# B&R Automation Studio project NAINV104C00R8L515F00 (part 16)

#### Visu_Page.typ - Change By Project
```iecst
(*2020-10-08*)
(**)
(*Page*)

TYPE
	tyUIP0000SSaver : 	STRUCT
		tySSaver : tyLyrP0000SSaver := (tyTxtMcStat:=(usiValueIdx:=3));
		tyMsgBoxHide : tyLyrC0008MsgBox := (tyBitmapIcon:=(uiRtStat:=1),tyBtnNo:=(uiRtStat:=1),tyBtnYes:=(uiRtStat:=1),tyLyr:=(uiRtStat:=1),tyTxtMsg:=(uiRtStat:=1),tyTxtTitle:=(uiRtStat:=1));
		tyMsgBoxLoginAsk : tyLyrC0008MsgBox := (tyBitmapIcon:=(usiValueIdx:=1),tyTxtTitle:=(usiValueIdx:=1),tyTxtMsg:=(usiValueIdx:=173),tyBtnYes:=(usiBitmapIdx:=1,usiTxtIdx:=3),tyBtnNo:=(usiBitmapIdx:=4,usiTxtIdx:=6),tyLyr:=(uiRtStat:=0));
	END_STRUCT;
END_TYPE

(**)

TYPE
	tyUIP0001Startup : 	STRUCT
		tyStartup : tyLyrP0001Startup;
		tyInitial : tyLyrP0001Initial;
		tyMsgBoxHide : tyLyrC0008MsgBox := (tyBitmapIcon:=(uiRtStat:=1),tyBtnNo:=(uiRtStat:=1),tyBtnYes:=(uiRtStat:=1),tyLyr:=(uiRtStat:=1),tyTxtMsg:=(uiRtStat:=1),tyTxtTitle:=(uiRtStat:=1));
		tyMsgBoxIPConfig : tyLyrC0008MsgBox := (tyBitmapIcon:=(usiValueIdx:=1),tyBtnNo:=(usiBitmapIdx:=3,usiTxtIdx:=2),tyBtnYes:=(usiBitmapIdx:=1,usiTxtIdx:=1),tyTxtTitle:=(usiValueIdx:=25));
	END_STRUCT;
END_TYPE

(**)

TYPE
	tyUIP0002Menu : 	STRUCT
		tyMenu : tyLyrP0002Menu := (tyBtnAlm:=(uiMaskRtStat:=0),tyBtnCommCtrl:=(uiMaskRtStat:=0),tyBtnGenInput:=(uiMaskRtStat:=0),tyBtnGenOutput:=(uiMaskRtStat:=0),tyBtnLang:=(uiMaskRtStat:=0),tyBtnLFCtrl:=(uiMaskRtStat:=0),tyBtnLFSet:=(uiMaskRtStat:=0),tyBtnMcInfo:=(uiMaskRtStat:=0),tyBtnMcSet:=(uiMaskRtStat:=0),tyBtnMnlRst:=(uiRtStat:=1),tyBtnMovCtrl:=(uiMaskRtStat:=0),tyBtnOpt:=(uiMaskRtStat:=0),tyBtnProdSel:=(uiMaskRtStat:=0),tyBtnProdSet:=(uiMaskRtStat:=0),tyBtnSimu:=(uiMaskRtStat:=0,uiRtStat:=1),tyBtnUsrMgmt:=(uiMaskRtStat:=0),tyGenMaskLyr:=(uiRtStat:=1),tySetMaskLyr:=(uiRtStat:=1));
		tyMsgBoxHide : tyLyrC0008MsgBox := (tyBitmapIcon:=(uiRtStat:=1),tyBtnNo:=(uiRtStat:=1),tyBtnYes:=(uiRtStat:=1),tyTxtMsg:=(uiRtStat:=1),tyTxtTitle:=(uiRtStat:=1),tyLyr:=(uiRtStat:=1));
		tyMsgBoxSelRcpWaitingBrd : tyLyrC0008MsgBox := (tyBitmapIcon:=(usiValueIdx:=1),tyTxtTitle:=(usiValueIdx:=2),tyTxtMsg:=(usiValueIdx:=100),tyBtnYes:=(uiRtStat:=1,usiBitmapIdx:=1,usiTxtIdx:=1),tyBtnNo:=(usiBitmapIdx:=1,usiTxtIdx:=3),tyLyr:=(uiRtStat:=0));
	END_STRUCT;
END_TYPE

(**)

TYPE
	tyUIP0100Login : 	STRUCT
		tyLogin : tyLyrP0100Login := (tyStringPw:=(sKeypadTitle:='Password'),tyStringUsrNm:=(sKeypadTitle:='User Name'));
		tyLogout : tyLyrP0100Logout := (tyLyr:=(uiRtStat:=1));
		tyMsgBoxHide : tyLyrC0008MsgBox := (tyBitmapIcon:=(uiRtStat:=1),tyBtnNo:=(uiRtStat:=1),tyBtnYes:=(uiRtStat:=1),tyTxtMsg:=(uiRtStat:=1),tyTxtTitle:=(uiRtStat:=1),tyLyr:=(uiRtStat:=1));
		tyMsgBoxNmNotExist : tyLyrC0008MsgBox := (tyBitmapIcon:=(usiValueIdx:=1),tyBtnNo:=(usiBitmapIdx:=1,usiTxtIdx:=3),tyBtnYes:=(uiRtStat:=1),tyLyr:=(uiRtStat:=0),tyTxtMsg:=(usiValueIdx:=23),tyTxtTitle:=(usiValueIdx:=1));
		tyMsgBoxPwMismatch : tyLyrC0008MsgBox := (tyBitmapIcon:=(usiValueIdx:=1),tyBtnNo:=(usiBitmapIdx:=1,usiTxtIdx:=3),tyBtnYes:=(uiRtStat:=1),tyLyr:=(uiRtStat:=0),tyTxtMsg:=(usiValueIdx:=24),tyTxtTitle:=(usiValueIdx:=1));
	END_STRUCT;
END_TYPE

(**)

TYPE
	tyUIP0200OpsGen : 	STRUCT
		tyOps : tyLyrP0200OpsGen := (tyBitmapDSCommIcon:=(uiMaskRtStat:=0),tyBitmapUSCommIcon:=(uiMaskRtStat:=0),tyBitmapRlsNewProd:=(uiRtStat:=1),tyBtnRlsNewProd:=(uiRtStat:=1));
		tyUSVSMEMA : tyLyrP0200OpsUSVSMEMA := (tyBtnUBAStat:=(uiRtStat:=1),tyBtnDual:=(uiRtStat:=1),tyLyr:=(uiRtStat:=1));
		tyDSVSMEMA : tyLyrP0200OpsDSVSMEMA := (tyBtnDSBStat:=(uiRtStat:=1),tyBtnDual:=(uiRtStat:=1),tyLyr:=(uiRtStat:=1));
		tyUSVSMEMA1 : tyLyrP0200OpsUSVSMEMA1 := (tyBtnUBAStat:=(uiRtStat:=1),tyBtnDual:=(uiRtStat:=1),tyLyr:=(uiRtStat:=1));
		tyDSVSMEMA1 : tyLyrP0200OpsDSVSMEMA1 := (tyBtnDSBStat:=(uiRtStat:=1),tyBtnDual:=(uiRtStat:=1),tyLyr:=(uiRtStat:=1));
		tyUSVSMEMA2 : tyLyrP0200OpsUSVSMEMA2 := (tyBtnUBAStat:=(uiRtStat:=1),tyBtnDual:=(uiRtStat:=1),tyLyr:=(uiRtStat:=1));
		tyBypsInitConv : tyLyrP0200OpsBypsInitConv := (tyLyr:=(uiRtStat:=1));
		tyMsgBoxHide : tyLyrC0008MsgBox := (tyBitmapIcon:=(uiRtStat:=1),tyBtnNo:=(uiRtStat:=1),tyBtnYes:=(uiRtStat:=1),tyTxtMsg:=(uiRtStat:=1),tyTxtTitle:=(uiRtStat:=1),tyLyr:=(uiRtStat:=1));
		tyMsgBoxRcpSelMsg : tyLyrC0008MsgBox;
		tyMsgBoxRstWaitingBrdAsk : tyLyrC0008MsgBox := (tyBitmapIcon:=(usiValueIdx:=1),tyTxtTitle:=(usiValueIdx:=23),tyTxtMsg:=(usiValueIdx:=125),tyBtnYes:=(usiBitmapIdx:=1,usiTxtIdx:=1),tyBtnNo:=(usiBitmapIdx:=3,usiTxtIdx:=2),tyLyr:=(uiRtStat:=0));
		tyRcyMsgHide : tyLyrC0010RcyMsg := (tyHotspotClose:=(uiRtStat:=1),tyLyr:=(uiRtStat:=1));
		tyRcyMsg : tyLyrC0010RcyMsg;
	END_STRUCT;
END_TYPE

(**)

TYPE
	tyUIP0201OpsConv : 	STRUCT
		tyOps : tyLyrP0201OpsConv := (tyBitmapRlsNewProd:=(uiRtStat:=1),tyBtnRlsNewProd:=(uiRtStat:=1));
		tyIOMonitor : tyLyrP0201OpsConvIOMonitor := (tyLyr:=(uiRtStat:=1));
		tyIOMonitorXStd : tyLyrP0201OpsConvIOMonitorXStd := (tyLyr:=(uiRtStat:=1));
		tyIOMonitorXStdMachineSafety : tyLyrP0201OpsConvIOMonitorMSafe;
		tyBypsInitConv : tyLyrP0200OpsBypsInitConv := (tyLyr:=(uiRtStat:=1));
		tyChgParam : tyLyrP0201OpsConvChgParam := (tyNumProdWidth:=(sKeypadTitle:='Product Width'),tyLyr:=(uiRtStat:=1));
		tyChgParamBkUp : tyLyrP0201OpsConvChgParam;
		tyNaviHide : tyLyrC0004Navi := (tyBtnLeft:=(uiRtStat:=1),tyBtnRgt:=(uiRtStat:=1),tyBtnBack:=(uiRtStat:=1));
		tyNaviBack : tyLyrC0004Navi := (tyBtnLeft:=(uiRtStat:=1),tyBtnRgt:=(uiRtStat:=1),tyBitmapPageDisp:=(uiRtStat:=1));
		tyMsgBoxHide : tyLyrC0008MsgBox := (tyBitmapIcon:=(uiRtStat:=1),tyBtnNo:=(uiRtStat:=1),tyBtnYes:=(uiRtStat:=1),tyTxtMsg:=(uiRtStat:=1),tyTxtTitle:=(uiRtStat:=1),tyLyr:=(uiRtStat:=1));
		tyMsgBoxSaveErr : tyLyrC0008MsgBox := (tyBitmapIcon:=(usiValueIdx:=1),tyTxtTitle:=(usiValueIdx:=7),tyTxtMsg:=(usiValueIdx:=71),tyBtnYes:=(uiRtStat:=1),tyBtnNo:=(usiBitmapIdx:=1,usiTxtIdx:=3));
		tyRcpPopUp : tyLyrC0012RcpPopUp := (tyLyr:=(uiRtStat:=1));
	END_STRUCT;
END_TYPE

(**)

TYPE
	tyUIP0300McInfo : 	STRUCT
		tyMcInfo : tyLyrP0300McInfo;
		tyMsgBoxHide : tyLyrC0008MsgBox := (tyBitmapIcon:=(uiRtStat:=1),tyTxtTitle:=(uiRtStat:=1),tyTxtMsg:=(uiRtStat:=1),tyBtnYes:=(uiRtStat:=1),tyBtnNo:=(uiRtStat:=1),tyLyr:=(uiRtStat:=1));
	END_STRUCT;
END_TYPE

(**)

TYPE
	tyUIP0400ProdSel : 	STRUCT
		tyProdSel : tyLyrP0400ProdSel := (tyStringSearch:=(sKeypadTitle:='Search Keyword'),tyTableRecipe:=(a_tyHotspot:=[(bRtCompl:=TRUE,bValue:=TRUE),14((0))],a_tyStringDataCol0:=[(sValue:='1'),(sValue:='2'),(sValue:='3'),(sValue:='4'),(sValue:='5'),(sValue:='6'),(sValue:='7'),(sValue:='8'),(sValue:='9'),2((sValue:='10')),4((0))],a_tyStringDataCol1:=[(usiColor:=1),14((0))],a_tyStringDataCol2:=[(usiColor:=1),14((0))],tyUISlider:=(iMaxValue:=1991,iMinValue:=1,iValue:=1),tyStringTitle0Col0Row0:=(sValue:='No'),tyStringTitle1Col1Row0:=(sValue:='Program Name'),tyStringTitle2Col2Row0:=(sValue:='Width')));
		tyRcpDet : tyLyrP0400RcpDet := (tyLyr:=(uiRtStat:=1));
		tyMsgBoxHide : tyLyrC0008MsgBox := (tyBitmapIcon:=(uiRtStat:=1),tyBtnNo:=(uiRtStat:=1),tyBtnYes:=(uiRtStat:=1),tyTxtMsg:=(uiRtStat:=1),tyTxtTitle:=(uiRtStat:=1),tyLyr:=(uiRtStat:=1));
		tyMsgBoxListErr : tyLyrC0008MsgBox := (tyBitmapIcon:=(usiValueIdx:=1),tyBtnNo:=(usiBitmapIdx:=1,usiTxtIdx:=3),tyBtnYes:=(uiRtStat:=1),tyLyr:=(uiRtStat:=0),tyTxtMsg:=(usiValueIdx:=42),tyTxtTitle:=(usiValueIdx:=2));
		tyMsgBoxRcpParamErr : tyLyrC0008MsgBox;
		tyMsgBoxLoadErr : tyLyrC0008MsgBox := (tyBitmapIcon:=(usiValueIdx:=1),tyBtnNo:=(usiBitmapIdx:=1,usiTxtIdx:=3),tyBtnYes:=(uiRtStat:=1),tyLyr:=(uiRtStat:=0),tyTxtMsg:=(usiValueIdx:=41),tyTxtTitle:=(usiValueIdx:=2));
		tyMsgBoxSelRcpAsk : tyLyrC0008MsgBox := (tyBitmapIcon:=(usiValueIdx:=1),tyBtnNo:=(usiBitmapIdx:=3,usiTxtIdx:=2),tyBtnYes:=(usiBitmapIdx:=1,usiTxtIdx:=1),tyLyr:=(uiRtStat:=0),tyTxtMsg:=(usiValueIdx:=43),tyTxtTitle:=(usiValueIdx:=2));
		tyMsgBoxSelRcpNoNm : tyLyrC0008MsgBox := (tyBitmapIcon:=(usiValueIdx:=1),tyBtnNo:=(usiBitmapIdx:=1,usiTxtIdx:=3),tyBtnYes:=(uiRtStat:=1),tyLyr:=(uiRtStat:=0),tyTxtMsg:=(usiValueIdx:=44),tyTxtTitle:=(usiValueIdx:=2));
		tyMsgBoxSaveErr : tyLyrC0008MsgBox := (tyBitmapIcon:=(usiValueIdx:=1),tyBtnNo:=(usiBitmapIdx:=1,usiTxtIdx:=3),tyBtnYes:=(uiRtStat:=1),tyLyr:=(uiRtStat:=0),tyTxtMsg:=(usiValueIdx:=71),tyTxtTitle:=(usiValueIdx:=2));
		tyMsgBoxGoToLFCtrlAsk : tyLyrC0008MsgBox := (tyBitmapIcon:=(usiValueIdx:=1),tyTxtTitle:=(usiValueIdx:=2),tyTxtMsg:=(usiValueIdx:=163),tyBtnYes:=(usiBitmapIdx:=1,usiTxtIdx:=1),tyBtnNo:=(usiBitmapIdx:=3,usiTxtIdx:=2),tyLyr:=(uiRtStat:=0));
		tyRcpPopUp : tyLyrC0012RcpPopUp := (tyLyr:=(uiRtStat:=1));
	END_STRUCT;
END_TYPE

(**)

TYPE
	tyUIP0600Alm : 	STRUCT
		tyAlm : tyLyrP0600Alm := (tyBtnCurr:=(bValue:=TRUE));
		tyMsgBoxHide : tyLyrC0008MsgBox := (tyBitmapIcon:=(uiRtStat:=1),tyBtnNo:=(uiRtStat:=1),tyBtnYes:=(uiRtStat:=1),tyTxtMsg:=(uiRtStat:=1),tyTxtTitle:=(uiRtStat:=1),tyLyr:=(uiRtStat:=1));
		tyRcyMsg : tyLyrC0010RcyMsg;
		tyRcyMsgHide : tyLyrC0010RcyMsg := (tyLyr:=(uiRtStat:=1));
		tyBtnCurr : tyUIBtn;
		tyBtnHistory : tyUIBtn;
		tyAlarm : tyUIAlarm;
	END_STRUCT;
END_TYPE

(**)

TYPE
	tyUIP0700LFCtrl : 	STRUCT
		tyLdr : tyLyrP0700LFCtrl := (tyBtnChgSeqAuto:=(uiMaskRtStat:=1),tyBtnChgSeqMnl:=(uiMaskRtStat:=1),tyTable1List:=(a_tyHotspot:=[(bRtCompl:=TRUE,bValue:=TRUE),14(0)],a_tyStringDataCol0:=[(sValue:='1'),(sValue:='2'),(sValue:='3'),(sValue:='4'),(sValue:='5'),(sValue:='6'),(sValue:='7'),(sValue:='8'),(sValue:='9'),(sValue:='10'),(sValue:='11'),(sValue:='12'),3((0))],a_tyStringDataCol1:=[0,14((0))],a_tyStringDataCol2:=[0,14((0))],a_tyStringDataCol4:=[(usiColor:=0),14((0))],a_tyTxtDataCol3:=[(usiColor:=1),14((0))],tyStringTitle0Col0Row0:=(sValue:='No'),tyStringTitle1Col1Row0:=(sValue:='Machine Name'),tyStringTitle2Col2Row0:=(sValue:='IP Address'),tyStringTitle3Col3Row0:=(sValue:='Status'),tyStringTitle4Col4Row0:=(sValue:='Recipe No'),tyUISlider:=(iMaxValue:=50,iMinValue:=1,iValue:=1,uiRtStat:=0)),tyLyr:=(uiRtStat:=0));
		tyMsgBoxHide : tyLyrC0008MsgBox := (tyBitmapIcon:=(uiRtStat:=1),tyBtnNo:=(uiRtStat:=1),tyBtnYes:=(uiRtStat:=1),tyTxtMsg:=(uiRtStat:=1),tyTxtTitle:=(uiRtStat:=1),tyLyr:=(uiRtStat:=1));
		tyMsgBoxChgAllAsk : tyLyrC0008MsgBox := (tyBitmapIcon:=(usiValueIdx:=1),tyTxtTitle:=(usiValueIdx:=9),tyTxtMsg:=(usiValueIdx:=156),tyBtnYes:=(usiBitmapIdx:=1,usiTxtIdx:=1),tyBtnNo:=(usiBitmapIdx:=3,usiTxtIdx:=2));
		tyMsgBoxChgSeqAutoAsk : tyLyrC0008MsgBox := (tyBitmapIcon:=(usiValueIdx:=1),tyTxtTitle:=(usiValueIdx:=9),tyTxtMsg:=(usiValueIdx:=157),tyBtnYes:=(usiBitmapIdx:=1,usiTxtIdx:=1),tyBtnNo:=(usiBitmapIdx:=3,usiTxtIdx:=2));
		tyMsgBoxChgSeqMnlAsk : tyLyrC0008MsgBox := (tyBitmapIcon:=(usiValueIdx:=1),tyTxtTitle:=(usiValueIdx:=9),tyTxtMsg:=(usiValueIdx:=158),tyBtnYes:=(usiBitmapIdx:=1,usiTxtIdx:=1),tyBtnNo:=(usiBitmapIdx:=3,usiTxtIdx:=2));
		tyMsgBoxSyncPLCTmAsk : tyLyrC0008MsgBox := (tyBitmapIcon:=(usiValueIdx:=1),tyTxtTitle:=(usiValueIdx:=9),tyTxtMsg:=(usiValueIdx:=159),tyBtnYes:=(usiBitmapIdx:=1,usiTxtIdx:=1),tyBtnNo:=(usiBitmapIdx:=3,usiTxtIdx:=2));
		tyMsgBoxTerminateOpsAsk : tyLyrC0008MsgBox := (tyBitmapIcon:=(usiValueIdx:=1),tyTxtTitle:=(usiValueIdx:=9),tyTxtMsg:=(usiValueIdx:=160),tyBtnYes:=(usiBitmapIdx:=1,usiTxtIdx:=1),tyBtnNo:=(usiBitmapIdx:=3,usiTxtIdx:=2));
		tyMsgBoxErrorAsk : tyLyrC0008MsgBox := (tyBitmapIcon:=(usiValueIdx:=1),tyTxtTitle:=(usiValueIdx:=9),tyTxtMsg:=(usiValueIdx:=165),tyBtnYes:=(uiRtStat:=1),tyBtnNo:=(usiBitmapIdx:=1,usiTxtIdx:=3));
	END_STRUCT;
END_TYPE

(**)

TYPE
	tyUIP0900GenIn : 	STRUCT
		tyGenIn : tyLyrP0900GenIn;
		tyMsgBoxHide : tyLyrC0008MsgBox := (tyBitmapIcon:=(uiRtStat:=1),tyBtnNo:=(uiRtStat:=1),tyBtnYes:=(uiRtStat:=1),tyTxtMsg:=(uiRtStat:=1),tyTxtTitle:=(uiRtStat:=1),tyLyr:=(uiRtStat:=1));
	END_STRUCT;
END_TYPE

(**)

TYPE
	tyUIP0910GenOut : 	STRUCT
		tyGenOut : tyLyrP0910GenOut;
		tyMsgBoxHide : tyLyrC0008MsgBox := (tyBitmapIcon:=(uiRtStat:=1),tyBtnNo:=(uiRtStat:=1),tyBtnYes:=(uiRtStat:=1),tyTxtMsg:=(uiRtStat:=1),tyTxtTitle:=(uiRtStat:=1),tyLyr:=(uiRtStat:=1));
	END_STRUCT;
END_TYPE

(**)

TYPE
	tyUIP0920MtrNPneuCtrl : 	STRUCT
		tyMtrNPneuCtrl : tyLyrP0920MtrNPneuCtrl;
		tyFullMaskHide : tyLyrC0002FullMask := (tyLyr:=(uiRtStat:=1));
		tyFullMaskEStop : tyLyrC0002FullMask := (tyBtnMask:=(usiTxtIdx:=20),tyLyr:=(uiRtStat:=0));
		tyFullMaskCWSig : tyLyrC0002FullMask := (tyBtnMask:=(usiTxtIdx:=21),tyLyr:=(uiRtStat:=0));
		tyFullMaskSafetyRly : tyLyrC0002FullMask := (tyBtnMask:=(usiTxtIdx:=12),tyLyr:=(uiRtStat:=0));
		tyMsgBoxHide : tyLyrC0008MsgBox := (tyBitmapIcon:=(uiRtStat:=1),tyBtnNo:=(uiRtStat:=1),tyBtnYes:=(uiRtStat:=1),tyTxtMsg:=(uiRtStat:=1),tyTxtTitle:=(uiRtStat:=1),tyLyr:=(uiRtStat:=1));
	END_STRUCT;
END_TYPE

(**)

TYPE
	tyUIP0921ClampNoRS : 	STRUCT
		tyCom : tyLyrP0921ClampNoRSCom;
		tyDC : tyLyrP0921ClampNoRSDC := (tyLyr:=(uiRtStat:=1));
		tyFB : tyLyrP0921ClampNoRSFB;
		tyFullMaskHide : tyLyrC0002FullMask := (tyLyr:=(uiRtStat:=1));
		tyFullMaskEStop : tyLyrC0002FullMask := (tyBtnMask:=(usiTxtIdx:=20),tyLyr:=(uiRtStat:=0));
		tyFullMaskCWSig : tyLyrC0002FullMask := (tyBtnMask:=(usiTxtIdx:=21),tyLyr:=(uiRtStat:=0));
		tyFullMaskSafetyRly : tyLyrC0002FullMask := (tyBtnMask:=(usiTxtIdx:=12),tyLyr:=(uiRtStat:=0));
		tyNaviBack : tyLyrC0004Navi := (tyBtnLeft:=(uiRtStat:=1),tyBtnRgt:=(uiRtStat:=1),tyBtnBack:=(uiRtStat:=0));
		tyMsgBoxHide : tyLyrC0008MsgBox := (tyBitmapIcon:=(uiRtStat:=1),tyBtnNo:=(uiRtStat:=1),tyBtnYes:=(uiRtStat:=1),tyTxtMsg:=(uiRtStat:=1),tyTxtTitle:=(uiRtStat:=1),tyLyr:=(uiRtStat:=1));
	END_STRUCT;
END_TYPE

(**)

TYPE
	tyUIP0922InletNOutletShutter : 	STRUCT
		tyInletShutterCom : tyLyrP0922InletShutterCom;
		tyInletShutterDC : tyLyrP0922InletShutterDC := (tyLyr:=(uiRtStat:=1));
		tyInletShutterFB : tyLyrP0922InletShutterFB;
		tyInletShutterDis : tyLyrP0922InletShutterDis := (tyLyr:=(uiRtStat:=1));
		tyOutletShutterCom : tyLyrP0922OutletShutterCom;
		tyOutletShutterDC : tyLyrP0922OutletShutterDC := (tyLyr:=(uiRtStat:=1));
		tyOutletShutterFB : tyLyrP0922OutletShutterFB;
		tyOutletShutterDis : tyLyrP0922OutletShutterDis := (tyLyr:=(uiRtStat:=1));
		tyDualMaskHide : tyLyrC0003DualMask := (tyLyr:=(uiRtStat:=1));
		tyDualMaskEStop : tyLyrC0003DualMask := (tyBtnLeftMask:=(uiMaskRtStat:=0,usiTxtIdx:=20),tyBtnRgtMask:=(uiMaskRtStat:=0,usiTxtIdx:=20));
		tyDualMaskCWSig : tyLyrC0003DualMask := (tyBtnLeftMask:=(uiMaskRtStat:=0,usiTxtIdx:=21),tyBtnRgtMask:=(uiMaskRtStat:=0,usiTxtIdx:=21));
		tyDualMaskSafetyRly : tyLyrC0003DualMask := (tyBtnLeftMask:=(uiMaskRtStat:=0,usiTxtIdx:=12),tyBtnRgtMask:=(uiMaskRtStat:=0,usiTxtIdx:=12));
		tyDualMaskAWMovInterrupt : tyLyrC0003DualMask := (tyBtnLeftMask:=(uiMaskRtStat:=0,usiTxtIdx:=17),tyBtnRgtMask:=(uiMaskRtStat:=0,usiTxtIdx:=17));
		tyNaviBack : tyLyrC0004Navi := (tyBtnLeft:=(uiRtStat:=1),tyBtnRgt:=(uiRtStat:=1),tyBtnBack:=(uiRtStat:=0));
		tyMsgBoxHide : tyLyrC0008MsgBox := (tyBitmapIcon:=(uiRtStat:=1),tyBtnNo:=(uiRtStat:=1),tyBtnYes:=(uiRtStat:=1),tyLyr:=(uiRtStat:=1),tyTxtMsg:=(uiRtStat:=1),tyTxtTitle:=(uiRtStat:=1));
	END_STRUCT;
END_TYPE

(**)

TYPE
	tyUIP0923Stopper : 	STRUCT
		tyCom : tyLyrP0923StopperCom;
		tyDC : tyLyrP0923StopperDC := (tyLyr:=(uiRtStat:=1));
		tyFB : tyLyrP0923StopperFB;
		tyFullMaskHide : tyLyrC0002FullMask := (tyLyr:=(uiRtStat:=1));
		tyFullMaskEStop : tyLyrC0002FullMask := (tyBtnMask:=(usiTxtIdx:=20),tyLyr:=(uiRtStat:=0));
		tyFullMaskCWSig : tyLyrC0002FullMask := (tyBtnMask:=(usiTxtIdx:=21),tyLyr:=(uiRtStat:=0));
		tyFullMaskSafetyRly : tyLyrC0002FullMask := (tyBtnMask:=(usiTxtIdx:=12),tyLyr:=(uiRtStat:=0));
		tyNaviBack : tyLyrC0004Navi := (tyBtnLeft:=(uiRtStat:=1),tyBtnRgt:=(uiRtStat:=1),tyBtnBack:=(uiRtStat:=0));
		tyMsgBoxHide : tyLyrC0008MsgBox := (tyBitmapIcon:=(uiRtStat:=1),tyBtnNo:=(uiRtStat:=1),tyBtnYes:=(uiRtStat:=1),tyTxtMsg:=(uiRtStat:=1),tyTxtTitle:=(uiRtStat:=1),tyLyr:=(uiRtStat:=1));
	END_STRUCT;
END_TYPE

(**)

TYPE
	tyUIP0924ClampWithRS : 	STRUCT
		tyClamp1WithRSCom : tyLyrP0924Clamp1WithRSCom;
		tyClamp1WithRSDC : tyLyrP0924Clamp1WithRSDC := (tyLyr:=(uiRtStat:=1));
		tyClamp1WithRSFB : tyLyrP0924Clamp1WithRSFB;
		tyClamp1WithRSDis : tyLyrP0924Clamp1WithRSDis := (tyLyr:=(uiRtStat:=1));
		tyClamp2WithRSCom : tyLyrP0924Clamp2WithRSCom;
		tyClamp2WithRSDC : tyLyrP0924Clamp2WithRSDC := (tyLyr:=(uiRtStat:=1));
		tyClamp2WithRSFB : tyLyrP0924Clamp2WithRSFB;
		tyClamp2WithRSDis : tyLyrP0924Clamp2WithRSDis := (tyLyr:=(uiRtStat:=1));
		tyClamp3WithRSCom : tyLyrP0924Clamp3WithRSCom;
		tyClamp3WithRSDC : tyLyrP0924Clamp3WithRSDC := (tyLyr:=(uiRtStat:=1));
		tyClamp3WithRSFB : tyLyrP0924Clamp3WithRSFB;
		tyClamp3WithRSDis : tyLyrP0924Clamp3WithRSDis := (tyLyr:=(uiRtStat:=1));
		tyDualMaskHide : tyLyrC0003DualMask := (tyLyr:=(uiRtStat:=1));
		tyDualMaskEStop : tyLyrC0003DualMask := (tyBtnLeftMask:=(uiMaskRtStat:=0,usiTxtIdx:=20),tyBtnRgtMask:=(uiMaskRtStat:=0,usiTxtIdx:=20));
		tyDualMaskCWSig : tyLyrC0003DualMask := (tyBtnLeftMask:=(uiMaskRtStat:=0,usiTxtIdx:=21),tyBtnRgtMask:=(uiMaskRtStat:=0,usiTxtIdx:=21));
		tyDualMaskSafetyRly : tyLyrC0003DualMask := (tyBtnLeftMask:=(uiMaskRtStat:=0,usiTxtIdx:=12),tyBtnRgtMask:=(uiMaskRtStat:=0,usiTxtIdx:=12));
		tyDualMaskAWMovInterrupt : tyLyrC0003DualMask := (tyBtnLeftMask:=(uiMaskRtStat:=0,usiTxtIdx:=17),tyBtnRgtMask:=(uiMaskRtStat:=0,usiTxtIdx:=17));
		tyNaviLyr1 : tyLyrC0004Navi := (tyBtnLeft:=(uiRtStat:=0),tyBtnRgt:=(uiRtStat:=0),tyBtnBack:=(uiRtStat:=0),tyBitmapPageDisp:=(uiRtStat:=0,usiValueIdx:=1));
		tyNaviLyr2 : tyLyrC0004Navi := (tyBtnLeft:=(uiRtStat:=0),tyBtnRgt:=(uiRtStat:=0),tyBtnBack:=(uiRtStat:=0),tyBitmapPageDisp:=(uiRtStat:=0,usiValueIdx:=2));
		tyMsgBoxHide : tyLyrC0008MsgBox := (tyBitmapIcon:=(uiRtStat:=1),tyBtnNo:=(uiRtStat:=1),tyBtnYes:=(uiRtStat:=1),tyLyr:=(uiRtStat:=1),tyTxtMsg:=(uiRtStat:=1),tyTxtTitle:=(uiRtStat:=1));
	END_STRUCT;
END_TYPE

(**)

TYPE
	tyUIP0931ConvInv : 	STRUCT
		tyConvCom : tyLyrP0931ConvCom;
		tyConvDC : tyLyrP0931ConvDC;
		tyConvFB : tyLyrP0931ConvFB := (tyBtnStop:=(bRtLk:=TRUE,bValue:=TRUE));
		tyInvCom : tyLyrP0931InvCom;
		tyInvDC : tyLyrP0931InvDC;
		tyInvFB : tyLyrP0931InvFB := (tyBtnStop:=(bRtLk:=TRUE,bValue:=TRUE));
		tyDualMaskHide : tyLyrC0003DualMask := (tyLyr:=(uiRtStat:=1));
		tyDualMaskEStop : tyLyrC0003DualMask := (tyBtnLeftMask:=(uiMaskRtStat:=0,usiTxtIdx:=20),tyBtnRgtMask:=(uiMaskRtStat:=0,usiTxtIdx:=20));
		tyDualMaskCWSig : tyLyrC0003DualMask := (tyBtnLeftMask:=(uiMaskRtStat:=0,usiTxtIdx:=21),tyBtnRgtMask:=(uiMaskRtStat:=0,usiTxtIdx:=21));
		tyDualMaskSafetyRly : tyLyrC0003DualMask := (tyBtnLeftMask:=(uiMaskRtStat:=0,usiTxtIdx:=12),tyBtnRgtMask:=(uiMaskRtStat:=0,usiTxtIdx:=12));
		tyDualMaskInletShutterInterrupt : tyLyrC0003DualMask := (tyBtnRgtMask:=(uiMaskRtStat:=0,usiTxtIdx:=27));
		tyDualMaskOutletShutterInterrupt : tyLyrC0003DualMask := (tyBtnRgtMask:=(uiMaskRtStat:=0,usiTxtIdx:=28));
		tyDualMaskInletNInvalid : tyLyrC0003DualMask := (tyBtnLeftMask:=(uiMaskRtStat:=0,usiTxtIdx:=23),tyBtnRgtMask:=(uiMaskRtStat:=0,usiTxtIdx:=27));
		tyDualMaskOutletNInvalid : tyLyrC0003DualMask := (tyBtnLeftMask:=(uiMaskRtStat:=0,usiTxtIdx:=23),tyBtnRgtMask:=(uiMaskRtStat:=0,usiTxtIdx:=28));
		tyDualMaskInvalidPos : tyLyrC0003DualMask := (tyBtnLeftMask:=(uiMaskRtStat:=0,usiTxtIdx:=23));
		tyDualMaskInvertInterrupt : tyLyrC0003DualMask := (tyBtnLeftMask:=(uiMaskRtStat:=1),tyBtnRgtMask:=(uiMaskRtStat:=0,usiTxtIdx:=29));
		tyDualMaskStopperInterruptInv : tyLyrC0003DualMask := (tyBtnLeftMask:=(uiMaskRtStat:=1),tyBtnRgtMask:=(uiMaskRtStat:=0,usiTxtIdx:=30));
		tyNaviBack : tyLyrC0004Navi := (tyBtnLeft:=(uiRtStat:=1),tyBtnRgt:=(uiRtStat:=1),tyBtnBack:=(uiRtStat:=0));
		tyMsgBoxHide : tyLyrC0008MsgBox := (tyBitmapIcon:=(uiRtStat:=1),tyBtnNo:=(uiRtStat:=1),tyBtnYes:=(uiRtStat:=1),tyTxtMsg:=(uiRtStat:=1),tyTxtTitle:=(uiRtStat:=1),tyLyr:=(uiRtStat:=1));
	END_STRUCT;
END_TYPE

(**)

TYPE
	tyUIP0934AW : 	STRUCT
		tyAW : tyLyrP0934AW := (tyNumNewWidth:=(sKeypadTitle:='New Width'));
		tyMotionStd : tyLyrC0001MotionStdAW := (tyBitmapMc:=(usiValueIdx:=2),tyBtnOpenLmtSen:=(usiTxtIdx:=3),tyBtnCloseLmtSen:=(usiTxtIdx:=1),tyBtnJogOpen:=(usiBitmapIdx:=2,usiTxtIdx:=2),tyBtnJogClose:=(usiBitmapIdx:=3,usiTxtIdx:=2),tyBtnStop:=(bValue:=TRUE),tyNumNomSpd:=(sKeypadTitle:='Normal Speed'),tyNumSlwSpd:=(sKeypadTitle:='Slow Speed'),tyNumStepSize:=(sKeypadTitle:='Step Size'),tyNumTargetPos:=(sKeypadTitle:='Target Position'));
		tyFullMaskHide : tyLyrC0002FullMask := (tyBtnMask:=(uiRtStat:=1),tyLyr:=(uiRtStat:=1));
		tyFullMaskEStop : tyLyrC0002FullMask := (tyBtnMask:=(usiTxtIdx:=20),tyLyr:=(uiRtStat:=0));
		tyFullMaskCWSig : tyLyrC0002FullMask := (tyBtnMask:=(usiTxtIdx:=21),tyLyr:=(uiRtStat:=0));
		tyFullMaskSafetyRly : tyLyrC0002FullMask := (tyBtnMask:=(usiTxtIdx:=12),tyLyr:=(uiRtStat:=0));
		tyFullMaskLftSenInterrupt : tyLyrC0002FullMask := (tyBtnMask:=(usiTxtIdx:=1),tyLyr:=(uiRtStat:=0));
		tyFullMaskRgtSenInterrupt : tyLyrC0002FullMask := (tyBtnMask:=(usiTxtIdx:=2),tyLyr:=(uiRtStat:=0));
		tyFullMaskInletShutterInterrupt : tyLyrC0002FullMask := (tyBtnMask:=(usiTxtIdx:=25),tyLyr:=(uiRtStat:=0));
		tyFullMaskOutletShutterInterrupt : tyLyrC0002FullMask := (tyBtnMask:=(usiTxtIdx:=26),tyLyr:=(uiRtStat:=0));
		tyFullMaskHomeSenInterrupt : tyLyrC0002FullMask := (tyBtnMask:=(usiTxtIdx:=23),tyLyr:=(uiRtStat:=0));
		tyFullMaskRemoteSenInterrupt : tyLyrC0002FullMask := (tyBtnMask:=(usiTxtIdx:=23),tyLyr:=(uiRtStat:=0));
		tyFullMaskInterrupt : tyLyrC0002FullMask := (tyBtnMask:=(usiTxtIdx:=26),tyLyr:=(uiRtStat:=0));
		tyNaviBack : tyLyrC0004Navi := (tyBtnLeft:=(uiRtStat:=1),tyBtnRgt:=(uiRtStat:=1),tyBtnBack:=(uiRtStat:=0));
		tyMsgBoxHide : tyLyrC0008MsgBox := (tyBitmapIcon:=(uiRtStat:=1),tyBtnNo:=(uiRtStat:=1),tyBtnYes:=(uiRtStat:=1),tyTxtMsg:=(uiRtStat:=1),tyTxtTitle:=(uiRtStat:=1),tyLyr:=(uiRtStat:=1));
	END_STRUCT;
END_TYPE

(**)

TYPE
	tyUIP0940CommCtrl : 	STRUCT
		tyUSSMEMA : tyLyrP0940CommCtrlUSSMEMA;
		tyDSSMEMA : tyLyrP0940CommCtrlDSSMEMA;
		tyUSSMEMA2 : tyLyrP0940CommCtrlUSSMEMA2;
		tyFullMaskHide : tyLyrC0002FullMask := (tyLyr:=(uiRtStat:=1));
		tyFullMaskEStop : tyLyrC0002FullMask := (tyBtnMask:=(usiTxtIdx:=20),tyLyr:=(uiRtStat:=0));
		tyFullMaskCWSig : tyLyrC0002FullMask := (tyBtnMask:=(usiTxtIdx:=21),tyLyr:=(uiRtStat:=0));
		tyFullMaskSafetyRly : tyLyrC0002FullMask := (tyBtnMask:=(usiTxtIdx:=12),tyLyr:=(uiRtStat:=0));
		tyMsgBoxHide : tyLyrC0008MsgBox := (tyBitmapIcon:=(uiRtStat:=1),tyBtnNo:=(uiRtStat:=1),tyBtnYes:=(uiRtStat:=1),tyTxtMsg:=(uiRtStat:=1),tyTxtTitle:=(uiRtStat:=1),tyLyr:=(uiRtStat:=1));
	END_STRUCT;
END_TYPE

(**)

TYPE
	tyUIP0950Simu : 	STRUCT
		tySimu : tyLyrP0950Simu;
		tyFullMaskHide : tyLyrC0002FullMask := (tyLyr:=(uiRtStat:=1));
		tyFullMaskEStop : tyLyrC0002FullMask := (tyBtnMask:=(usiTxtIdx:=1));
		tyFullMaskCWSig : tyLyrC0002FullMask := (tyBtnMask:=(usiTxtIdx:=2));
		tyFullMaskSafetyRly : tyLyrC0002FullMask := (tyBtnMask:=(usiTxtIdx:=3));
		tyMsgBoxHide : tyLyrC0008MsgBox := (tyBitmapIcon:=(uiRtStat:=1),tyBtnNo:=(uiRtStat:=1),tyBtnYes:=(uiRtStat:=1),tyTxtMsg:=(uiRtStat:=1),tyTxtTitle:=(uiRtStat:=1),tyLyr:=(uiRtStat:=1));
	END_STRUCT;
END_TYPE

(**)

TYPE
	tyUIP1000Lang : 	STRUCT
		tyLang : tyLyrP1000Lang := (tyBtnEnglish:=(bRtLk:=TRUE,bValue:=TRUE),tyNumYear:=(sKeypadTitle:='Year'),tyNumMonth:=(sKeypadTitle:='Month'),tyNumDay:=(sKeypadTitle:='Day'),tyNumHour:=(sKeypadTitle:='Hour'),tyNumMinute:=(sKeypadTitle:='Minute'),tyNumSecond:=(sKeypadTitle:='Second'));
		tyLangBkUp : tyLyrP1000Lang;
		tyMsgBoxHide : tyLyrC0008MsgBox := (tyBitmapIcon:=(uiRtStat:=1),tyBtnNo:=(uiRtStat:=1),tyBtnYes:=(uiRtStat:=1),tyTxtMsg:=(uiRtStat:=1),tyTxtTitle:=(uiRtStat:=1),tyLyr:=(uiRtStat:=1));
		tyMsgBoxSaveErr : tyLyrC0008MsgBox := (tyBitmapIcon:=(usiValueIdx:=1),tyBtnNo:=(usiBitmapIdx:=1,usiTxtIdx:=3),tyBtnYes:=(uiRtStat:=1),tyLyr:=(uiRtStat:=0),tyTxtMsg:=(usiValueIdx:=65),tyTxtTitle:=(usiValueIdx:=20));
	END_STRUCT;
END_TYPE

(**)

TYPE
	tyUIP1020McSetNavi : 	STRUCT
		tyNavi : tyLyrP1020McSetNavi;
		tyMsgBoxHide : tyLyrC0008MsgBox := (tyBitmapIcon:=(uiRtStat:=1),tyBtnNo:=(uiRtStat:=1),tyBtnYes:=(uiRtStat:=1),tyTxtMsg:=(uiRtStat:=1),tyTxtTitle:=(uiRtStat:=1),tyLyr:=(uiRtStat:=1));
	END_STRUCT;
END_TYPE

(**)

TYPE
	tyUIP1021McSetGen : 	STRUCT
		tyGen : tyLyrP1021McSetGen := (tyDrpDnDefaultMcMod:=(usiValueMaxIdx:=1),tyDrpDnDefaultFlippedBrd:=(usiValueMaxIdx:=2),tyNumConvInitTm:=(sKeypadTitle:='Conveyor Initialize Time'),tyNumTranInErrDlyTm:=(sKeypadTitle:='Transfer In Error Dly Tm'),tyNumTranOutErrDlyTm:=(sKeypadTitle:='Transfer Out Error Dly Tm'),tyNumWidthAtHm:=(sKeypadTitle:='Width At Home Position'),tyNumWidthOffset:=(sKeypadTitle:='Width Offset'),tyStringMcNm:=(sKeypadTitle:='Machine Name'),tyNumSSaverTm:=(sKeypadTitle:='Screen Saver Time'),tyStringSubnetMask:=(sKeypadTitle:='Subnet Mask'),tyStringIPAddr:=(sKeypadTitle:='IP Address'),tyNumStopperAtLftPos:=(sKeypadTitle:='Stopper At Left Pos'),tyNumStopperAtRgtPos:=(sKeypadTitle:='Stopper At Right Pos'));
		tyGenBkUp : tyLyrP1021McSetGen;
		tyNetwork : tyLyrP1021McSetNetwork := (tyStringIPAddr:=(sKeypadTitle:='IP Address'),tyStringSubnetMask:=(sKeypadTitle:='Subnet Mask'),tyLyr:=(uiRtStat:=1));
		tyNaviLyr1 : tyLyrC0004Navi := (tyBtnLeft:=(uiRtStat:=0),tyBtnRgt:=(uiRtStat:=0),tyBtnBack:=(uiRtStat:=0),tyBitmapPageDisp:=(uiRtStat:=0,usiValueIdx:=1));
		tyNaviLyr2 : tyLyrC0004Navi := (tyBtnLeft:=(uiRtStat:=0),tyBtnRgt:=(uiRtStat:=0),tyBtnBack:=(uiRtStat:=0),tyBitmapPageDisp:=(uiRtStat:=0,usiValueIdx:=2));
		tyMsgBoxHide : tyLyrC0008MsgBox := (tyBitmapIcon:=(uiRtStat:=1),tyBtnNo:=(uiRtStat:=1),tyBtnYes:=(uiRtStat:=1),tyTxtMsg:=(uiRtStat:=1),tyTxtTitle:=(uiRtStat:=1),tyLyr:=(uiRtStat:=1));
		tyMsgBoxExitAsk : tyLyrC0008MsgBox := (tyBitmapIcon:=(usiValueIdx:=1),tyBtnNo:=(usiBitmapIdx:=3,usiTxtIdx:=2),tyBtnYes:=(usiBitmapIdx:=1,usiTxtIdx:=1),tyTxtMsg:=(usiValueIdx:=70),tyTxtTitle:=(usiValueIdx:=14),tyLyr:=(uiRtStat:=0));
		tyMsgBoxSaveErr : tyLyrC0008MsgBox := (tyBitmapIcon:=(usiValueIdx:=1),tyBtnNo:=(usiBitmapIdx:=1,usiTxtIdx:=3),tyBtnYes:=(uiRtStat:=1),tyTxtMsg:=(usiValueIdx:=71),tyTxtTitle:=(usiValueIdx:=14));
		tyMsgBoxUpdtSubnetAsk : tyLyrC0008MsgBox := (tyBitmapIcon:=(usiValueIdx:=1),tyBtnNo:=(usiBitmapIdx:=3,usiTxtIdx:=2),tyBtnYes:=(usiBitmapIdx:=1,usiTxtIdx:=1),tyTxtMsg:=(usiValueIdx:=75),tyTxtTitle:=(usiValueIdx:=14));
		tyMsgBoxUpdtSubnetErr : tyLyrC0008MsgBox := (tyBitmapIcon:=(usiValueIdx:=1),tyBtnNo:=(usiBitmapIdx:=1,usiTxtIdx:=3),tyBtnYes:=(uiRtStat:=1),tyTxtMsg:=(usiValueIdx:=76),tyTxtTitle:=(usiValueIdx:=14));
		tyMsgBoxSubnetInvalid : tyLyrC0008MsgBox := (tyBitmapIcon:=(usiValueIdx:=1),tyBtnNo:=(usiBitmapIdx:=1,usiTxtIdx:=3),tyBtnYes:=(uiRtStat:=1),tyTxtMsg:=(usiValueIdx:=77),tyTxtTitle:=(usiValueIdx:=14));
		tyMsgBoxUpdtIPAddrAsk : tyLyrC0008MsgBox := (tyBitmapIcon:=(usiValueIdx:=1),tyBtnNo:=(usiBitmapIdx:=3,usiTxtIdx:=2),tyBtnYes:=(usiBitmapIdx:=1,usiTxtIdx:=1),tyTxtMsg:=(usiValueIdx:=72),tyTxtTitle:=(usiValueIdx:=14));
		tyMsgBoxUpdtIPAddrErr : tyLyrC0008MsgBox := (tyBitmapIcon:=(usiValueIdx:=1),tyBtnNo:=(usiBitmapIdx:=1,usiTxtIdx:=3),tyBtnYes:=(uiRtStat:=1),tyTxtMsg:=(usiValueIdx:=73),tyTxtTitle:=(usiValueIdx:=14));
		tyMsgBoxIPAddrInvalid : tyLyrC0008MsgBox := (tyBitmapIcon:=(usiValueIdx:=1),tyBtnNo:=(usiBitmapIdx:=1,usiTxtIdx:=3),tyBtnYes:=(uiRtStat:=1),tyTxtMsg:=(usiValueIdx:=74),tyTxtTitle:=(usiValueIdx:=14));
		tyMsgBoxChgNetworkAsk : tyLyrC0008MsgBox := (tyBitmapIcon:=(usiValueIdx:=1),tyBtnNo:=(usiBitmapIdx:=3,usiTxtIdx:=2),tyBtnYes:=(usiBitmapIdx:=1,usiTxtIdx:=1),tyTxtTitle:=(usiValueIdx:=14));
		tyMsgBoxIPAddrInvalidEdit : tyLyrC0008MsgBox := (tyBitmapIcon:=(usiValueIdx:=1),tyTxtTitle:=(usiValueIdx:=14),tyTxtMsg:=(usiValueIdx:=184),tyBtnYes:=(uiRtStat:=1),tyBtnNo:=(usiBitmapIdx:=1,usiTxtIdx:=3));
		tyMsgBoxSubnetInvalidEdit : tyLyrC0008MsgBox := (tyBitmapIcon:=(usiValueIdx:=1),tyTxtTitle:=(usiValueIdx:=14),tyTxtMsg:=(usiValueIdx:=185),tyBtnYes:=(uiRtStat:=1),tyBtnNo:=(usiBitmapIdx:=1,usiTxtIdx:=3));
		tyMsgBoxGetIPAddrErr : tyLyrC0008MsgBox := (tyBitmapIcon:=(usiValueIdx:=1),tyTxtTitle:=(usiValueIdx:=14),tyTxtMsg:=(usiValueIdx:=186),tyBtnYes:=(uiRtStat:=1),tyBtnNo:=(usiBitmapIdx:=1,usiTxtIdx:=3));
		tyMsgBoxGetSubnetErr : tyLyrC0008MsgBox := (tyBitmapIcon:=(usiValueIdx:=1),tyTxtTitle:=(usiValueIdx:=14),tyTxtMsg:=(usiValueIdx:=187),tyBtnYes:=(uiRtStat:=1),tyBtnNo:=(usiBitmapIdx:=1,usiTxtIdx:=3));
		tyMsgBoxSetDHCPError : tyLyrC0008MsgBox := (tyBitmapIcon:=(usiValueIdx:=1),tyTxtTitle:=(usiValueIdx:=14),tyTxtMsg:=(usiValueIdx:=188),tyBtnYes:=(uiRtStat:=1),tyBtnNo:=(usiBitmapIdx:=1,usiTxtIdx:=3));
	END_STRUCT;
END_TYPE

(**)

TYPE
	tyUIP1022McSetVComm : 	STRUCT
		tyVComSel : tyLyrP1022McSetVCommSel;
		tyVComSelBkUp : tyLyrP1022McSetVCommSel;
		tyLF : tyLyrP1022McSetVCommLF;
		tyLFBkUp : tyLyrP1022McSetVCommLF;
		tyVComSvy : tyLyrP1022McSetVCommSvy := (tyNumSndAliveTm:=(diValueMax:=1800000,diValueMin:=5000,sKeypadTitle:='Send Alive Tm'),tyNumSvySystemPort:=(diValueMin:=65535,sKeypadTitle:='System Port'),tyLyr:=(uiRtStat:=1));
		tyVComSvyBkUp : tyLyrP1022McSetVCommSvy;
		tyNaviLyr1 : tyLyrC0004Navi := (tyBtnLeft:=(uiRtStat:=1),tyBtnRgt:=(uiRtStat:=1),tyBtnBack:=(uiRtStat:=0),tyBitmapPageDisp:=(uiRtStat:=1,usiValueIdx:=0),tyLyr:=(uiRtStat:=0));
		tyNaviLyr2 : tyLyrC0004Navi := (tyBtnLeft:=(uiRtStat:=1),tyBtnRgt:=(uiRtStat:=1),tyBtnBack:=(uiRtStat:=0),tyBitmapPageDisp:=(uiRtStat:=1,usiValueIdx:=1),tyLyr:=(uiRtStat:=0));
		tyNaviLyr3 : tyLyrC0004Navi := (tyBtnLeft:=(uiRtStat:=0),tyBtnRgt:=(uiRtStat:=0),tyBtnBack:=(uiRtStat:=0),tyBitmapPageDisp:=(uiRtStat:=0,usiValueIdx:=0));
		tyNaviLyr4 : tyLyrC0004Navi := (tyBtnLeft:=(uiRtStat:=0),tyBtnRgt:=(uiRtStat:=0),tyBtnBack:=(uiRtStat:=0),tyBitmapPageDisp:=(uiRtStat:=0,usiValueIdx:=0));
		tyNaviBack : tyLyrC0004Navi := (tyBtnLeft:=(uiRtStat:=1),tyBtnRgt:=(uiRtStat:=1),tyBtnBack:=(uiRtStat:=0));
		tyMsgBoxHide : tyLyrC0008MsgBox := (tyBitmapIcon:=(uiRtStat:=1),tyBtnNo:=(uiRtStat:=1),tyBtnYes:=(uiRtStat:=1),tyTxtMsg:=(uiRtStat:=1),tyTxtTitle:=(uiRtStat:=1),tyLyr:=(uiRtStat:=1));
		tyMsgBoxExitAsk : tyLyrC0008MsgBox := (tyBitmapIcon:=(usiValueIdx:=1),tyBtnNo:=(usiBitmapIdx:=3,usiTxtIdx:=2),tyBtnYes:=(usiBitmapIdx:=1,usiTxtIdx:=1),tyLyr:=(uiRtStat:=0),tyTxtMsg:=(usiValueIdx:=70),tyTxtTitle:=(usiValueIdx:=16));
		tyMsgBoxSaveErr : tyLyrC0008MsgBox;
	END_STRUCT;
END_TYPE

(**)

TYPE
	tyUIP1023McSetHComm : 	STRUCT
		tyGen : tyLyrP1023McSetHCommGen := (tyLyr:=(uiRtStat:=1));
		tyUSSel : tyLyrP1023McSetHCommSel := (tyBtnSMEMA:=(bRtLk:=TRUE,bValue:=TRUE));
		tyUSSMEMA : tyLyrP1023McSetHCommSMEMA := (tyDrpDnSMEMAMod:=(usiValueMaxIdx:=1),tyLyr:=(uiRtStat:=1));
		tyUSHermes : tyLyrP1023McSetHCommUSHermes := (tyNumSndAliveTm:=(diValueMax:=1800000,diValueMin:=5000,sKeypadTitle:='Send Alive Time'),tyNumLaneID:=(diValueMax:=1000,diValueMin:=1,sKeypadTitle:='Lane ID'),tyNumHostPort:=(diValueMax:=65535,sKeypadTitle:='Host Port'),tyStringHostAddr:=(sKeypadTitle:='Host Address'));
		tyDSSel : tyLyrP1023McSetHCommSel := (tyBtnSMEMA:=(bRtLk:=TRUE,bValue:=TRUE),tyLyr:=(uiRtStat:=1));
		tyDSSel2 : tyLyrP1023McSetHCommSel := (tyBtnSMEMA:=(bRtLk:=TRUE,bValue:=TRUE),tyLyr:=(uiRtStat:=1));
		tyDSSMEMA : tyLyrP1023McSetHCommSMEMA := (tyDrpDnSMEMAMod:=(usiValueMaxIdx:=1),tyLyr:=(uiRtStat:=1));
		tyDSSMEMA2 : tyLyrP1023McSetHCommSMEMA := (tyDrpDnSMEMAMod:=(usiValueMaxIdx:=1),tyLyr:=(uiRtStat:=1));
		tyDSHermes : tyLyrP1023McSetHCommDSHermes := (tyNumLaneID:=(diValueMax:=1000,diValueMin:=1,sKeypadTitle:='Lane ID'),tyNumSvrPort:=(diValueMax:=65535,sKeypadTitle:='Server Port'),tyNumSndAliveTm:=(diValueMax:=1800000,diValueMin:=5000,sKeypadTitle:='Send Alive Time'));
		tyDSHermes2 : tyLyrP1023McSetHCommDSHermes := (tyNumLaneID:=(diValueMax:=1000,diValueMin:=1,sKeypadTitle:='Lane ID'),tyNumSvrPort:=(diValueMax:=65535,sKeypadTitle:='Server Port'),tyNumSndAliveTm:=(diValueMax:=1800000,diValueMin:=5000,sKeypadTitle:='Send Alive Time'));
		tyUSSelBkUp : tyLyrP1023McSetHCommSel;
		tyUSSMEMABkUp : tyLyrP1023McSetHCommSMEMA;
		tyUSHermesBkUp : tyLyrP1023McSetHCommUSHermes;
		tyDSSelBkUp : tyLyrP1023McSetHCommSel;
		tyDSSelBkUp2 : tyLyrP1023McSetHCommSel;
		tyDSSMEMABkUp : tyLyrP1023McSetHCommSMEMA;
		tyDSSMEMABkUp2 : tyLyrP1023McSetHCommSMEMA;
		tyDSHermesBkUp : tyLyrP1023McSetHCommDSHermes;
		tyDSHermesBkUp2 : tyLyrP1023McSetHCommDSHermes;
		tyUSSel2 : tyLyrP1023McSetHCommSel := (tyBtnSMEMA:=(bRtLk:=TRUE,bValue:=TRUE));
		tyUSSMEMA2 : tyLyrP1023McSetHCommSMEMA := (tyDrpDnSMEMAMod:=(usiValueMaxIdx:=1),tyLyr:=(uiRtStat:=1));
		tyUSHermes2 : tyLyrP1023McSetHCommUSHermes := (tyNumSndAliveTm:=(diValueMax:=1800000,diValueMin:=5000,sKeypadTitle:='Send Alive Time'),tyNumLaneID:=(diValueMax:=1000,diValueMin:=1,sKeypadTitle:='Lane ID'),tyNumHostPort:=(diValueMax:=65535,sKeypadTitle:='Host Port'),tyStringHostAddr:=(sKeypadTitle:='Host Address'));
		tyUSSelBkUp2 : tyLyrP1023McSetHCommSel;
		tyUSSMEMABkUp2 : tyLyrP1023McSetHCommSMEMA;
		tyUSHermesBkUp2 : tyLyrP1023McSetHCommUSHermes;
		tyNaviLyr1 : tyLyrC0004Navi := (tyBtnLeft:=(uiRtStat:=0),tyBtnRgt:=(uiRtStat:=0),tyBtnBack:=(uiRtStat:=0),tyBitmapPageDisp:=(uiRtStat:=0,usiValueIdx:=1));
		tyNaviLyr2 : tyLyrC0004Navi := (tyBtnLeft:=(uiRtStat:=0),tyBtnRgt:=(uiRtStat:=0),tyBtnBack:=(uiRtStat:=0),tyBitmapPageDisp:=(uiRtStat:=0,usiValueIdx:=2));
		tyMsgBoxHide : tyLyrC0008MsgBox := (tyBitmapIcon:=(uiRtStat:=1),tyBtnNo:=(uiRtStat:=1),tyBtnYes:=(uiRtStat:=1),tyTxtMsg:=(uiRtStat:=1),tyTxtTitle:=(uiRtStat:=1),tyLyr:=(uiRtStat:=1));
		tyMsgBoxExitAsk : tyLyrC0008MsgBox := (tyBitmapIcon:=(usiValueIdx:=1),tyBtnNo:=(usiBitmapIdx:=3,usiTxtIdx:=2),tyBtnYes:=(usiBitmapIdx:=1,usiTxtIdx:=1),tyLyr:=(uiRtStat:=0),tyTxtMsg:=(usiValueIdx:=70),tyTxtTitle:=(usiValueIdx:=16));
		tyMsgBoxSaveErr : tyLyrC0008MsgBox := (tyBitmapIcon:=(usiValueIdx:=1),tyBtnNo:=(usiBitmapIdx:=1,usiTxtIdx:=3),tyBtnYes:=(uiRtStat:=1),tyLyr:=(uiRtStat:=0),tyTxtMsg:=(usiValueIdx:=71),tyTxtTitle:=(usiValueIdx:=15));
		tyMsgBoxIPAddrInvalid : tyLyrC0008MsgBox := (tyBitmapIcon:=(usiValueIdx:=1),tyBtnNo:=(usiBitmapIdx:=1,usiTxtIdx:=3),tyBtnYes:=(uiRtStat:=1),tyLyr:=(uiRtStat:=0),tyTxtMsg:=(usiValueIdx:=74),tyTxtTitle:=(usiValueIdx:=14));
	END_STRUCT;
END_TYPE

(**)

TYPE
	tyUIP1024McSetAntiGap : 	STRUCT
		tyAntiGap : tyLyrP1024McSetAntiGap := (tyNumLftSenOff:=(sKeypadTitle:='Left Sensor Signal'),tyNumRgtSenOff:=(sKeypadTitle:='Right Sensor Signal'));
		tyAntiGapBkUp : tyLyrP1024McSetAntiGap;
		tyMsgBoxHide : tyLyrC0008MsgBox := (tyBitmapIcon:=(uiRtStat:=1),tyBtnNo:=(uiRtStat:=1),tyBtnYes:=(uiRtStat:=1),tyTxtMsg:=(uiRtStat:=1),tyTxtTitle:=(uiRtStat:=1),tyLyr:=(uiRtStat:=1));
		tyMsgBoxExitAsk : tyLyrC0008MsgBox := (tyBitmapIcon:=(usiValueIdx:=1),tyBtnNo:=(usiBitmapIdx:=3,usiTxtIdx:=2),tyBtnYes:=(usiBitmapIdx:=1,usiTxtIdx:=1),tyLyr:=(uiRtStat:=0),tyTxtMsg:=(usiValueIdx:=70),tyTxtTitle:=(usiValueIdx:=17));
		tyMsgBoxSaveErr : tyLyrC0008MsgBox := (tyBitmapIcon:=(usiValueIdx:=1),tyBtnNo:=(usiBitmapIdx:=1,usiTxtIdx:=3),tyBtnYes:=(uiRtStat:=1),tyTxtMsg:=(usiValueIdx:=71),tyTxtTitle:=(usiValueIdx:=17));
		tyNaviBack : tyLyrC0004Navi := (tyBtnLeft:=(uiRtStat:=1),tyBtnRgt:=(uiRtStat:=1),tyBtnBack:=(uiRtStat:=0));
	END_STRUCT;
END_TYPE

(**)

TYPE
	tyUIP1026McSetTeach : 	STRUCT
		tyTeachStopperAtLftPos : tyLyrP1026McSetTeach := (tyBtnGet:=(usiTxtIdx:=200),tyBtnGo:=(usiTxtIdx:=201));
		tyTeachStopperAtRgtPos : tyLyrP1026McSetTeach := (tyBtnGet:=(usiTxtIdx:=202),tyBtnGo:=(usiTxtIdx:=203));
		tyMotionStd : tyLyrC0001MotionStdInvert := (tyBitmapMc:=(usiValueIdx:=2),tyBtnHmLmtSen:=(usiTxtIdx:=4),tyBtnRmtLmtSen:=(usiTxtIdx:=4),tyBtnJogHm:=(usiTxtIdx:=4),tyBtnJogRmt:=(usiBitmapIdx:=1,usiTxtIdx:=4),tyNumNomSpd:=(sKeypadTitle:='Normal Speed'),tyNumSlwSpd:=(sKeypadTitle:='Slow Speed'),tyNumStepSize:=(sKeypadTitle:='Step Size'),tyNumTargetPos:=(sKeypadTitle:='Target Position'));
		tyFullMaskHide : tyLyrC0002FullMask := (tyBtnMask:=(uiRtStat:=1),tyLyr:=(uiRtStat:=1));
		tyFullMaskEStop : tyLyrC0002FullMask := (tyBtnMask:=(usiTxtIdx:=20),tyLyr:=(uiRtStat:=0));
		tyFullMaskCWSig : tyLyrC0002FullMask := (tyBtnMask:=(usiTxtIdx:=21),tyLyr:=(uiRtStat:=0));
		tyFullMaskSafetyRly : tyLyrC0002FullMask := (tyBtnMask:=(usiTxtIdx:=12),tyLyr:=(uiRtStat:=0));
		tyNaviBack : tyLyrC0004Navi := (tyBtnLeft:=(uiRtStat:=1),tyBtnRgt:=(uiRtStat:=1),tyBtnBack:=(uiRtStat:=0));
		tyMsgBoxHide : tyLyrC0008MsgBox := (tyBitmapIcon:=(uiRtStat:=1),tyBtnNo:=(uiRtStat:=1),tyBtnYes:=(uiRtStat:=1),tyTxtMsg:=(uiRtStat:=1),tyTxtTitle:=(uiRtStat:=1),tyLyr:=(uiRtStat:=1));
		tyMsgBoxUpdtStopperAtLftPos : tyLyrC0008MsgBox := (tyBitmapIcon:=(usiValueIdx:=1),tyTxtTitle:=(usiValueIdx:=22),tyTxtMsg:=(usiValueIdx:=85),tyBtnYes:=(uiRtStat:=1,usiBitmapIdx:=1,usiTxtIdx:=1),tyBtnNo:=(usiBitmapIdx:=1,usiTxtIdx:=3));
		tyMsgBoxUpdtStopperAtRgtPos : tyLyrC0008MsgBox := (tyBitmapIcon:=(usiValueIdx:=1),tyTxtTitle:=(usiValueIdx:=22),tyTxtMsg:=(usiValueIdx:=86),tyBtnYes:=(uiRtStat:=1,usiBitmapIdx:=1,usiTxtIdx:=1),tyBtnNo:=(usiBitmapIdx:=1,usiTxtIdx:=3));
	END_STRUCT;
END_TYPE

(**)

TYPE
	tyUIP1040ProdSet : 	STRUCT
		tyProdSet : tyLyrP1040ProdSet := (tyBtnSave:=(uiMaskRtStat:=0),tyNumProdWidth:=(sKeypadTitle:='Product Width'),tyStringRecipeNm:=(sKeypadTitle:='Recipe Name'),tyStringSearch:=(sKeypadTitle:='Search Keyword'),tyTableRecipe:=(a_tyHotspot:=[(bRtCompl:=TRUE,bValue:=TRUE),14((0))],a_tyStringDataCol0:=[(sValue:='1'),(sValue:='2'),(sValue:='3'),(sValue:='4'),(sValue:='5'),(sValue:='6'),(sValue:='7'),(sValue:='8'),(sValue:='9'),(sValue:='10'),5((0))],a_tyStringDataCol1:=[(usiColor:=1),14(0)],a_tyStringDataCol2:=[(usiColor:=1),14(0)],tyUISlider:=(iMaxValue:=2000,iMinValue:=1,iValue:=1),tyStringTitle0Col0Row0:=(sValue:='No'),tyStringTitle1Col1Row0:=(sValue:='Product Name'),tyStringTitle2Col2Row0:=(sValue:='Width'),uiMaskRtStat:=1),tyDrpDnMcMode:=(usiValueMaxIdx:=1),tyDrpDnFlippedBrd:=(usiValueMaxIdx:=2),tyStringMatchCode:=(sKeypadTitle:='Match Code'));
		tyMsgBoxHide : tyLyrC0008MsgBox := (tyBitmapIcon:=(uiRtStat:=1),tyBtnNo:=(uiRtStat:=1),tyBtnYes:=(uiRtStat:=1),tyTxtMsg:=(uiRtStat:=1),tyTxtTitle:=(uiRtStat:=1),tyLyr:=(uiRtStat:=1));
		tyMsgBoxSaveAsk : tyLyrC0008MsgBox := (tyBitmapIcon:=(usiValueIdx:=1),tyBtnNo:=(usiBitmapIdx:=3,usiTxtIdx:=2),tyBtnYes:=(usiBitmapIdx:=1,usiTxtIdx:=1),tyLyr:=(uiRtStat:=0),tyTxtMsg:=(usiValueIdx:=46),tyTxtTitle:=(usiValueIdx:=8));
		tyMsgBoxSaveErr : tyLyrC0008MsgBox := (tyBitmapIcon:=(usiValueIdx:=1),tyBtnNo:=(usiBitmapIdx:=1,usiTxtIdx:=3),tyBtnYes:=(uiRtStat:=1),tyLyr:=(uiRtStat:=0),tyTxtMsg:=(usiValueIdx:=40),tyTxtTitle:=(usiValueIdx:=8));
		tyMsgBoxListFull : tyLyrC0008MsgBox := (tyBitmapIcon:=(usiValueIdx:=1),tyBtnNo:=(usiBitmapIdx:=1,usiTxtIdx:=3),tyBtnYes:=(uiRtStat:=1),tyLyr:=(uiRtStat:=0),tyTxtMsg:=(usiValueIdx:=59),tyTxtTitle:=(usiValueIdx:=8));
		tyMsgBoxListErr : tyLyrC0008MsgBox := (tyBitmapIcon:=(usiValueIdx:=1),tyBtnNo:=(usiBitmapIdx:=1,usiTxtIdx:=3),tyBtnYes:=(uiRtStat:=1),tyLyr:=(uiRtStat:=0),tyTxtMsg:=(usiValueIdx:=42),tyTxtTitle:=(usiValueIdx:=8));
		tyMsgBoxSaveNoNm : tyLyrC0008MsgBox := (tyBitmapIcon:=(usiValueIdx:=1),tyBtnNo:=(usiBitmapIdx:=1,usiTxtIdx:=3),tyBtnYes:=(uiRtStat:=1),tyLyr:=(uiRtStat:=0),tyTxtMsg:=(usiValueIdx:=47),tyTxtTitle:=(usiValueIdx:=8));
		tyMsgBoxReloadCurrRcp : tyLyrC0008MsgBox := (tyBitmapIcon:=(usiValueIdx:=1),tyBtnNo:=(usiBitmapIdx:=1,usiTxtIdx:=3),tyBtnYes:=(uiRtStat:=1),tyLyr:=(uiRtStat:=0),tyTxtMsg:=(usiValueIdx:=50),tyTxtTitle:=(usiValueIdx:=8));
		tyMsgBoxDelCurrRcpAsk : tyLyrC0008MsgBox := (tyBitmapIcon:=(usiValueIdx:=1),tyBtnNo:=(usiBitmapIdx:=1,usiTxtIdx:=3),tyBtnYes:=(uiRtStat:=1),tyLyr:=(uiRtStat:=0),tyTxtMsg:=(usiValueIdx:=51),tyTxtTitle:=(usiValueIdx:=8));
		tyMsgBoxDelNmNotExist : tyLyrC0008MsgBox := (tyBitmapIcon:=(usiValueIdx:=1),tyBtnNo:=(usiBitmapIdx:=1,usiTxtIdx:=3),tyBtnYes:=(uiRtStat:=1),tyLyr:=(uiRtStat:=0),tyTxtMsg:=(usiValueIdx:=54),tyTxtTitle:=(usiValueIdx:=8));
		tyMsgBoxDelNmEmpty : tyLyrC0008MsgBox := (tyBitmapIcon:=(usiValueIdx:=1),tyBtnNo:=(usiBitmapIdx:=1,usiTxtIdx:=3),tyBtnYes:=(uiRtStat:=1),tyLyr:=(uiRtStat:=0),tyTxtMsg:=(usiValueIdx:=60),tyTxtTitle:=(usiValueIdx:=8));
		tyMsgBoxDelErr : tyLyrC0008MsgBox := (tyBitmapIcon:=(usiValueIdx:=1),tyBtnNo:=(usiBitmapIdx:=1,usiTxtIdx:=3),tyBtnYes:=(uiRtStat:=1),tyLyr:=(uiRtStat:=0),tyTxtMsg:=(usiValueIdx:=52),tyTxtTitle:=(usiValueIdx:=8));
		tyMsgBoxDelAsk : tyLyrC0008MsgBox := (tyBitmapIcon:=(usiValueIdx:=1),tyBtnNo:=(usiBitmapIdx:=3,usiTxtIdx:=2),tyBtnYes:=(usiBitmapIdx:=1,usiTxtIdx:=1),tyLyr:=(uiRtStat:=0),tyTxtMsg:=(usiValueIdx:=53),tyTxtTitle:=(usiValueIdx:=8));
		tyMsgBoxToXMLAsk : tyLyrC0008MsgBox := (tyBitmapIcon:=(usiValueIdx:=1),tyTxtTitle:=(usiValueIdx:=8),tyTxtMsg:=(usiValueIdx:=61),tyBtnYes:=(usiBitmapIdx:=1,usiTxtIdx:=1),tyBtnNo:=(usiBitmapIdx:=3,usiTxtIdx:=2),tyLyr:=(uiRtStat:=0));
		tyMsgBoxToXMLErr : tyLyrC0008MsgBox := (tyBitmapIcon:=(usiValueIdx:=1),tyTxtTitle:=(usiValueIdx:=8),tyTxtMsg:=(usiValueIdx:=62),tyBtnYes:=(uiRtStat:=1),tyBtnNo:=(usiBitmapIdx:=1,usiTxtIdx:=3),tyLyr:=(uiRtStat:=0));
		tyMsgBoxFromXMLAsk : tyLyrC0008MsgBox := (tyBitmapIcon:=(usiValueIdx:=1),tyTxtTitle:=(usiValueIdx:=8),tyTxtMsg:=(usiValueIdx:=63),tyBtnYes:=(usiBitmapIdx:=1,usiTxtIdx:=1),tyBtnNo:=(usiBitmapIdx:=3,usiTxtIdx:=2),tyLyr:=(uiRtStat:=0));
		tyMsgBoxFromXMLErr : tyLyrC0008MsgBox := (tyBitmapIcon:=(usiValueIdx:=1),tyTxtTitle:=(usiValueIdx:=8),tyTxtMsg:=(usiValueIdx:=64),tyBtnYes:=(uiRtStat:=1),tyBtnNo:=(usiBitmapIdx:=1,usiTxtIdx:=3),tyLyr:=(uiRtStat:=0));
		tyMsgBoxSaveListErr : tyLyrC0008MsgBox := (tyBitmapIcon:=(usiValueIdx:=1),tyTxtTitle:=(usiValueIdx:=8),tyTxtMsg:=(usiValueIdx:=66),tyBtnYes:=(uiRtStat:=1),tyBtnNo:=(usiBitmapIdx:=1,usiTxtIdx:=3),tyLyr:=(uiRtStat:=0));
		tyRcpPopUp : tyLyrC0012RcpPopUp := (tyLyr:=(uiRtStat:=1));
	END_STRUCT;
END_TYPE

(**)

TYPE
	tyUIP1050LFSet : 	STRUCT
		tyLdr : tyLyrP1050LFSetLdr := (tyTable1List:=(a_tyHotspot:=[(bRtCompl:=TRUE,bValue:=TRUE),14(0)],a_tyStringDataCol0:=[(sValue:='1'),(sValue:='2'),(sValue:='3'),(sValue:='4'),(sValue:='5'),(sValue:='6'),(sValue:='7'),(sValue:='8'),(sValue:='9'),(sValue:='10'),(sValue:='11'),(sValue:='12'),(sValue:='13'),(sValue:='14'),(sValue:='15')],a_tyStringDataCol1:=[(usiColor:=1),14(0)],a_tyStringDataCol2:=[(usiColor:=1),14(0)],a_tyTxtDataCol3:=[(usiColor:=1),14(0)],tyStringTitle0Col0Row0:=(sValue:='No'),tyStringTitle1Col1Row0:=(sValue:='Machine Name'),tyStringTitle2Col2Row0:=(sValue:='IP Address'),tyStringTitle3Col3Row0:=(sValue:='Status'),tyUISlider:=(iMaxValue:=c_diLFClntNum-c_uiP1050TableSize+1,iMinValue:=1,iValue:=1)),tyNumBeforeOven:=(sKeypadTitle:='Machine Index Before Oven 1'),tyNumBeforeOven2:=(sKeypadTitle:='Machine Index Before Oven 2'),tyNumAfterOven:=(sKeypadTitle:='Machine Index After Oven 1'),tyNumAfterOven2:=(sKeypadTitle:='Machine Index After Oven 2'));
		tyLdrEdit : tyLyrP1050LFSetLdrEdit := (tyStringIPAddr:=(sKeypadTitle:='IP Address'),tyTxtLblInfoThirdParty:=(uiRtStat:=1),tyLyr:=(uiRtStat:=1));
		tyLdrBkUp : tyLyrP1050LFSetLdr;
		tyMsgBoxHide : tyLyrC0008MsgBox := (tyBitmapIcon:=(uiRtStat:=1),tyTxtTitle:=(uiRtStat:=1),tyTxtMsg:=(uiRtStat:=1),tyBtnYes:=(uiRtStat:=1),tyBtnNo:=(uiRtStat:=1),tyLyr:=(uiRtStat:=1));
		tyMsgBoxSaveErr : tyLyrC0008MsgBox := (tyBitmapIcon:=(usiValueIdx:=1),tyTxtTitle:=(usiValueIdx:=9),tyTxtMsg:=(usiValueIdx:=71),tyBtnYes:=(uiRtStat:=1),tyBtnNo:=(usiBitmapIdx:=1,usiTxtIdx:=3),tyLyr:=(uiRtStat:=0));
		tyMsgBoxDelAsk : tyLyrC0008MsgBox := (tyBitmapIcon:=(usiValueIdx:=1),tyTxtTitle:=(usiValueIdx:=9),tyTxtMsg:=(usiValueIdx:=153),tyBtnYes:=(usiBitmapIdx:=1,usiTxtIdx:=1),tyBtnNo:=(usiBitmapIdx:=3,usiTxtIdx:=2),tyLyr:=(uiRtStat:=0));
		tyMsgBoxIPAddrInvalid : tyLyrC0008MsgBox := (tyBitmapIcon:=(usiValueIdx:=1),tyTxtTitle:=(usiValueIdx:=9),tyTxtMsg:=(usiValueIdx:=155),tyBtnYes:=(uiRtStat:=1),tyBtnNo:=(usiBitmapIdx:=1,usiTxtIdx:=3),tyLyr:=(uiRtStat:=0));
		tyMsgBoxIPAddrDuplicate : tyLyrC0008MsgBox := (tyBitmapIcon:=(usiValueIdx:=1),tyTxtTitle:=(usiValueIdx:=9),tyTxtMsg:=(usiValueIdx:=163),tyBtnYes:=(uiRtStat:=1),tyBtnNo:=(usiBitmapIdx:=1,usiTxtIdx:=3),tyLyr:=(uiRtStat:=0));
	END_STRUCT;
END_TYPE

(**)

TYPE
	tyUIP1080UsrMgmt : 	STRUCT
		tyActHide : tyLyrP1080UsrMgmtAct := (tyLyr:=(uiRtStat:=1));
		tyEdit : tyLyrP1080UsrMgmtAct := (tyStringPw:=(sKeypadTitle:='Password'),tyStringUsrNm:=(uiMaskRtStat:=0));
		tyCreate : tyLyrP1080UsrMgmtAct := (tyStringPw:=(sKeypadTitle:='Password'),tyStringUsrNm:=(sKeypadTitle:='User Name'));
		tyUsrMgmt : tyLyrP1080UsrMgmt := (tyTableList:=(a_tyHotspot:=[11((bRtCompl:=TRUE,bValue:=TRUE)),4((0))],a_tyStringDataCol0:=[(sValue:='1'),(sValue:='2'),(sValue:='3'),(sValue:='4'),(sValue:='5'),(sValue:='6'),(sValue:='7'),(sValue:='8'),(sValue:='9'),(sValue:='10'),(sValue:='11'),4((0))],a_tyStringDataCol1:=[(usiColor:=1),8((0)),2(0),4((0))],a_tyStringDataCol2:=[0,14((0))],a_tyTxtDataCol3:=[(usiColor:=1),8((0)),2(0),4((0))],tyStringTitle0Col0Row0:=(sValue:='No'),tyStringTitle1Col1Row0:=(sValue:='Username'),tyStringTitle3Col3Row0:=(sValue:='Level Title'),uiMaskRtStat:=1));
		tyMsgBoxHide : tyLyrC0008MsgBox := (tyBitmapIcon:=(uiRtStat:=1),tyBtnNo:=(uiRtStat:=1),tyBtnYes:=(uiRtStat:=1),tyTxtMsg:=(uiRtStat:=1),tyTxtTitle:=(uiRtStat:=1),tyLyr:=(uiRtStat:=1));
		tyMsgBoxAddErr : tyLyrC0008MsgBox := (tyBitmapIcon:=(usiValueIdx:=1),tyBtnNo:=(usiBitmapIdx:=1,usiTxtIdx:=3),tyBtnYes:=(uiRtStat:=1),tyLyr:=(uiRtStat:=0),tyTxtMsg:=(usiValueIdx:=27),tyTxtTitle:=(usiValueIdx:=1));
		tyMsgBoxEditErr : tyLyrC0008MsgBox := (tyBitmapIcon:=(usiValueIdx:=1),tyBtnNo:=(usiBitmapIdx:=1,usiTxtIdx:=3),tyBtnYes:=(uiRtStat:=1),tyLyr:=(uiRtStat:=0),tyTxtMsg:=(usiValueIdx:=28),tyTxtTitle:=(usiValueIdx:=1));
		tyMsgBoxAddNmExist : tyLyrC0008MsgBox := (tyBitmapIcon:=(usiValueIdx:=1),tyBtnNo:=(usiBitmapIdx:=1,usiTxtIdx:=3),tyBtnYes:=(uiRtStat:=1),tyLyr:=(uiRtStat:=0),tyTxtMsg:=(usiValueIdx:=22),tyTxtTitle:=(usiValueIdx:=1));
		tyMsgBoxEditParamErr : tyLyrC0008MsgBox := (tyBitmapIcon:=(usiValueIdx:=1),tyBtnNo:=(usiBitmapIdx:=1,usiTxtIdx:=3),tyBtnYes:=(uiRtStat:=1),tyLyr:=(uiRtStat:=0),tyTxtMsg:=(usiValueIdx:=24),tyTxtTitle:=(usiValueIdx:=1));
		tyMsgBoxAddParamErr : tyLyrC0008MsgBox := (tyBitmapIcon:=(usiValueIdx:=1),tyBtnNo:=(usiBitmapIdx:=1,usiTxtIdx:=3),tyBtnYes:=(uiRtStat:=1),tyLyr:=(uiRtStat:=0),tyTxtMsg:=(usiValueIdx:=21),tyTxtTitle:=(usiValueIdx:=1));
		tyMsgBoxListFull : tyLyrC0008MsgBox := (tyBitmapIcon:=(usiValueIdx:=1),tyBtnNo:=(usiBitmapIdx:=1,usiTxtIdx:=3),tyBtnYes:=(uiRtStat:=1),tyLyr:=(uiRtStat:=0),tyTxtMsg:=(usiValueIdx:=35),tyTxtTitle:=(usiValueIdx:=1));
		tyMsgBoxDelNmNotExist : tyLyrC0008MsgBox := (tyBitmapIcon:=(usiValueIdx:=1),tyBtnNo:=(usiBitmapIdx:=1,usiTxtIdx:=3),tyBtnYes:=(uiRtStat:=1),tyLyr:=(uiRtStat:=0),tyTxtMsg:=(usiValueIdx:=37),tyTxtTitle:=(usiValueIdx:=1));
		tyMsgBoxDelParamErr : tyLyrC0008MsgBox := (tyBitmapIcon:=(usiValueIdx:=1),tyBtnNo:=(usiBitmapIdx:=1,usiTxtIdx:=3),tyBtnYes:=(uiRtStat:=1),tyLyr:=(uiRtStat:=0),tyTxtMsg:=(usiValueIdx:=31),tyTxtTitle:=(usiValueIdx:=1));
		tyMsgBoxDelLastAdminErr : tyLyrC0008MsgBox := (tyBitmapIcon:=(usiValueIdx:=1),tyBtnNo:=(usiBitmapIdx:=1,usiTxtIdx:=3),tyBtnYes:=(uiRtStat:=1),tyLyr:=(uiRtStat:=0),tyTxtMsg:=(usiValueIdx:=26),tyTxtTitle:=(usiValueIdx:=1));
		tyMsgBoxDelAsk : tyLyrC0008MsgBox := (tyBitmapIcon:=(usiValueIdx:=1),tyBtnNo:=(usiBitmapIdx:=3,usiTxtIdx:=2),tyBtnYes:=(usiBitmapIdx:=1,usiTxtIdx:=1),tyLyr:=(uiRtStat:=0),tyTxtMsg:=(usiValueIdx:=25),tyTxtTitle:=(usiValueIdx:=1));
		tyMsgBoxDelErr : tyLyrC0008MsgBox := (tyBitmapIcon:=(usiValueIdx:=1),tyBtnNo:=(usiBitmapIdx:=1,usiTxtIdx:=3),tyBtnYes:=(uiRtStat:=1),tyLyr:=(uiRtStat:=0),tyTxtMsg:=(usiValueIdx:=30),tyTxtTitle:=(usiValueIdx:=1));
	END_STRUCT;
END_TYPE

(**)

TYPE
	tyUIP1081UsrAccessRgt : 	STRUCT
		tyUsrAccessRgtSel : tyLyrP1081UsrMgmtUsrAccessRgtSel := (tyDrpDnLevel:=(usiValueMaxIdx:=2));
		tyUsrAccessRgtLvl1 : tyLyrP1081UsrMgmtUsrAccessRgt := (tyStringNm:=(sKeypadTitle:='Level Name'),tyTxtTitle:=(usiValueIdx:=0));
		tyUsrAccessRgtLvl2 : tyLyrP1081UsrMgmtUsrAccessRgt := (tyStringNm:=(sKeypadTitle:='Level Name'),tyTxtTitle:=(usiValueIdx:=1));
		tyUsrAccessRgtLvl3 : tyLyrP1081UsrMgmtUsrAccessRgt := (tyStringNm:=(sKeypadTitle:='Level Name'),tyTxtTitle:=(usiValueIdx:=2));
		tyUsrAccessRgtLvl1BkUp : tyLyrP1081UsrMgmtUsrAccessRgt;
		tyUsrAccessRgtLvl2BkUp : tyLyrP1081UsrMgmtUsrAccessRgt;
		tyUsrAccessRgtLvl3BkUp : tyLyrP1081UsrMgmtUsrAccessRgt;
		tyNaviBack : tyLyrC0004Navi := (tyBtnLeft:=(uiRtStat:=1),tyBtnRgt:=(uiRtStat:=1),tyBtnBack:=(uiRtStat:=0));
		tyMsgBoxHide : tyLyrC0008MsgBox := (tyBitmapIcon:=(uiRtStat:=1),tyBtnNo:=(uiRtStat:=1),tyBtnYes:=(uiRtStat:=1),tyTxtMsg:=(uiRtStat:=1),tyTxtTitle:=(uiRtStat:=1),tyLyr:=(uiRtStat:=1));
		tyMsgBoxExitAsk : tyLyrC0008MsgBox := (tyBitmapIcon:=(usiValueIdx:=1),tyBtnNo:=(usiBitmapIdx:=3,usiTxtIdx:=2),tyBtnYes:=(usiBitmapIdx:=1,usiTxtIdx:=1),tyLyr:=(uiRtStat:=0),tyTxtMsg:=(usiValueIdx:=70),tyTxtTitle:=(usiValueIdx:=1));
		tyMsgBoxSaveErr : tyLyrC0008MsgBox := (tyBitmapIcon:=(usiValueIdx:=1),tyBtnNo:=(usiBitmapIdx:=1,usiTxtIdx:=3),tyBtnYes:=(uiRtStat:=1),tyLyr:=(uiRtStat:=0),tyTxtMsg:=(usiValueIdx:=34),tyTxtTitle:=(usiValueIdx:=1));
	END_STRUCT;
END_TYPE

(**)
(*Common Layers*)

TYPE
	tyUICom : 	STRUCT
		tyMain : tyLyrC0005Main := (tyBtnStep:=(uiRtStat:=1),tyBtnReset:=(uiMaskRtStat:=0),tyBtnStop:=(uiMaskRtStat:=0));
		tySet : tyLyrC0006Set := (tyBtnSave:=(uiMaskRtStat:=0));
		tyNotif : tyLyrC0007Notif := (tyLyr:=(uiRtStat:=1));
		tyInfo : tyLyrC0009Info := (tyLyr:=(uiRtStat:=1));
		tyLoading : tyLyrC0011Loading := (tyLyr:=(uiRtStat:=1));
	END_STRUCT;
END_TYPE

(**)
(*Visu Property*)

TYPE
	tyUIProperty : 	STRUCT
		tyVisu : tyVisu;
		tyKeypad : tyKeypad;
		tyUITxtSnippets : tyTxtSnippets;
	END_STRUCT;
END_TYPE
```

#### Visu_Page.var - Change By Project
```iecst
(*2020-10-08*)
(**)
(*UI Constant*)
VAR CONSTANT
	c_uiC0007TableSize : UINT := 4;
	c_uiP0200TableSize : UINT := 6;
	c_uiP0400TableSize : UINT := 10;
	c_uiP0600TableSize : UINT := 18;
	c_uiP0700TableSize : UINT := 11;
	c_uiP1040TableSize : UINT := 10;
	c_uiP1050TableSize : UINT := 12;
	c_uiP1080TableSize : UINT := 11;
END_VAR
(**)
(*Page*)
VAR
	tyP0000SSaver : tyUIP0000SSaver; (*Screen Saver*)
END_VAR
(**)
VAR
	tyP0001Startup : tyUIP0001Startup; (*Startup*)
END_VAR
(**)
VAR
	tyP0002Menu : tyUIP0002Menu; (*Menu*)
END_VAR
(**)
VAR
	tyP0100Login : tyUIP0100Login; (*Login*)
END_VAR
(**)
VAR
	tyP0200OpsGen : tyUIP0200OpsGen; (*Operation*)
END_VAR
(**)
VAR
	tyP0201OpsConv : tyUIP0201OpsConv; (*Operation*)
END_VAR
(**)
VAR
	tyP0300McInfo : tyUIP0300McInfo; (*Operation*)
END_VAR
(**)
VAR
	tyP0400ProdSel : tyUIP0400ProdSel; (*Product Selection*)
END_VAR
(**)
VAR
	tyP0600Alm : tyUIP0600Alm; (*Alarm*)
END_VAR
(**)
VAR
	tyP0700LFCtrl : tyUIP0700LFCtrl; (*Lead Follow*)
END_VAR
(**)
VAR
	tyP0900GenIn : tyUIP0900GenIn; (*General Input*)
END_VAR
(**)
VAR
	tyP0910GenOut : tyUIP0910GenOut; (*General Output*)
END_VAR
(**)
VAR
	tyP0920MtrNPneuCtrl : tyUIP0920MtrNPneuCtrl; (*Motor And Pneumatic Control*)
END_VAR
(**)
VAR
	tyP0921ClampNoRS : tyUIP0921ClampNoRS; (*Clamp*)
END_VAR
(**)
VAR
	tyP0922InletNOutletShutter : tyUIP0922InletNOutletShutter; (*Flipper*)
END_VAR
(**)
VAR
	tyP0923Stopper : tyUIP0923Stopper; (*Stopper*)
END_VAR
(**)
VAR
	tyP0924ClampWithRS : tyUIP0924ClampWithRS; (*Clamp1 and Clamp2*)
END_VAR
(**)
VAR
	tyP0931ConvInv : tyUIP0931ConvInv; (*Conveyor & Inverter*)
END_VAR
(**)
VAR
	tyP0934AW : tyUIP0934AW; (*Auto Width*)
END_VAR
(**)
VAR
	tyP0940CommCtrl : tyUIP0940CommCtrl; (*Communication Control*)
END_VAR
(**)
VAR
	tyP0950Simu : tyUIP0950Simu; (*Simulation*)
END_VAR
(**)
VAR
	tyP1000Lang : tyUIP1000Lang; (*Language & Time*)
END_VAR
(**)
VAR
	tyP1020McSetNavi : tyUIP1020McSetNavi; (*Machine Setting - Navigation*)
END_VAR
(**)
VAR
	tyP1021McSetGen : tyUIP1021McSetGen; (*Machine Setting - General*)
END_VAR
(**)
VAR
	tyP1022McSetVComm : tyUIP1022McSetVComm; (*Machine Setting - Commnunication*)
END_VAR
(**)
VAR
	tyP1023McSetHComm : tyUIP1023McSetHComm; (*Machine Setting - Commnunication*)
END_VAR
(**)
VAR
	tyP1024McSetAntiGap : tyUIP1024McSetAntiGap; (*Machine Setting - Anti Gap Sensor*)
END_VAR
(**)
VAR
	tyP1026McSetTeach : tyUIP1026McSetTeach; (*Machine Setting - Teach*)
END_VAR
(**)
VAR
	tyP1040ProdSet : tyUIP1040ProdSet; (*Product Setting*)
END_VAR
(**)
VAR
	tyP1050LFSet : tyUIP1050LFSet; (*Leader Follower Setting*)
END_VAR
(**)
VAR
	tyP1080UsrMgmt : tyUIP1080UsrMgmt; (*User Management*)
END_VAR
(**)
VAR
	tyP1081UsrMgmtUsrAccessRgt : tyUIP1081UsrAccessRgt; (*User Managemen User Access*)
END_VAR
(**)
(*Common*)
VAR
	tyCommon : tyUICom;
END_VAR
(**)
(*UI Property*)
VAR
	tyProperty : tyUIProperty; (*Visualization Properties*)
END_VAR
```

#### Visu_Layer.typ - Change By Project
```iecst
(*2020-10-08*)
(**)
(*Common Layer*)

TYPE
	tyLyrC0001MotionStd : 	STRUCT
		tyBitmapOrigin : tyUIBitmap;
		tyBitmapPwr : tyUIBitmap;
		tyBitmapRst : tyUIBitmap;
		tyBitmapStop : tyUIBitmap;
		tyBitmapMc : tyUIBitmap;
		tyBtnPosLmtSen : tyUIBtn;
		tyBtnNegLmtSen : tyUIBtn;
		tyBtnJogPos : tyUIBtn;
		tyBtnJogNeg : tyUIBtn;
		tyBtnMovAbs : tyUIBtn;
		tyBtnMovRel : tyUIBtn;
		tyBtnOrigin : tyUIBtn;
		tyBtnPwr : tyUIBtn;
		tyBtnRst : tyUIBtn;
		tyBtnStop : tyUIBtn;
		tyNumCurrPos : tyUINum;
		tyNumErrCode : tyUINum;
		tyNumNomSpd : tyUINum;
		tyNumSlwSpd : tyUINum;
		tyNumStepSize : tyUINum;
		tyNumTargetPos : tyUINum;
		tyStringStat : tyUILString;
		tyLyr : tyUILyr;
	END_STRUCT;
	tyLyrC0001MotionStdAW : 	STRUCT
		tyBitmapOrigin : tyUIBitmap;
		tyBitmapPwr : tyUIBitmap;
		tyBitmapRst : tyUIBitmap;
		tyBitmapStop : tyUIBitmap;
		tyBitmapMc : tyUIBitmap;
		tyBtnOpenLmtSen : tyUIBtn;
		tyBtnCloseLmtSen : tyUIBtn;
		tyBtnJogOpen : tyUIBtn;
		tyBtnJogClose : tyUIBtn;
		tyBtnMovAbs : tyUIBtn;
		tyBtnMovRel : tyUIBtn;
		tyBtnOrigin : tyUIBtn;
		tyBtnPwr : tyUIBtn;
		tyBtnRst : tyUIBtn;
		tyBtnStop : tyUIBtn;
		tyNumCurrPos : tyUINum;
		tyNumErrCode : tyUINum;
		tyNumNomSpd : tyUINum;
		tyNumSlwSpd : tyUINum;
		tyNumStepSize : tyUINum;
		tyNumTargetPos : tyUINum;
		tyStringStat : tyUILString;
		tyLyr : tyUILyr;
	END_STRUCT;
	tyLyrC0001MotionStdInvert : 	STRUCT
		tyBitmapOrigin : tyUIBitmap;
		tyBitmapPwr : tyUIBitmap;
		tyBitmapRst : tyUIBitmap;
		tyBitmapStop : tyUIBitmap;
		tyBitmapMc : tyUIBitmap;
		tyBtnHmLmtSen : tyUIBtn;
		tyBtnRmtLmtSen : tyUIBtn;
		tyBtnJogHm : tyUIBtn;
		tyBtnJogRmt : tyUIBtn;
		tyBtnMovAbs : tyUIBtn;
		tyBtnMovRel : tyUIBtn;
		tyBtnOrigin : tyUIBtn;
		tyBtnPwr : tyUIBtn;
		tyBtnRst : tyUIBtn;
		tyBtnStop : tyUIBtn;
		tyNumCurrPos : tyUINum;
		tyNumErrCode : tyUINum;
		tyNumNomSpd : tyUINum;
		tyNumSlwSpd : tyUINum;
		tyNumStepSize : tyUINum;
		tyNumTargetPos : tyUINum;
		tyStringStat : tyUILString;
		tyLyr : tyUILyr;
	END_STRUCT;
	tyLyrC0002FullMask : 	STRUCT
		tyBtnMask : tyUIBtn;
		tyLyr : tyUILyr;
	END_STRUCT;
	tyLyrC0003DualMask : 	STRUCT
		tyBtnLeftMask : tyUIBtn;
		tyBtnRgtMask : tyUIBtn;
		tyLyr : tyUILyr;
	END_STRUCT;
	tyLyrC0004Navi : 	STRUCT
		tyBtnLeft : tyUIBtn;
		tyBtnRgt : tyUIBtn;
		tyBtnBack : tyUIBtn;
		tyBitmapPageDisp : tyUIBitmap;
		tyLyr : tyUILyr;
	END_STRUCT;
	tyLyrC0005Main : 	STRUCT
		tyBtnHome : tyUIBtn;
		tyBtnNotification : tyUIBtn;
		tyBtnStart : tyUIBtn;
		tyBtnStop : tyUIBtn;
		tyBtnStep : tyUIBtn;
		tyBtnReset : tyUIBtn;
		tyBitmapStatBar : tyUIBitmap;
		tyBtnMuteBuz : tyUIBtn := (uiMaskRtStat:=0);
		tyHotspotNaviStart : tyUIHotspot;
		tyBtnAlarm : tyUIBtn;
	END_STRUCT;
	tyLyrC0006Set : 	STRUCT
		tyBtnSave : tyUIBtn;
		tyLyr : tyUILyr;
	END_STRUCT;
	tyLyrC0007Notif : 	STRUCT
		tyTxtUsrLv : tyUITxt;
		tyTxtLFMc : tyUITxt;
		tyStringUsrNm : tyUIString;
		tyHotspotClose : tyUIHotspot;
		tyHotspotShowInfo : tyUIHotspot;
		tyBitmapShowInfo : tyUIBitmap;
		tyLyr : tyUILyr;
	END_STRUCT;
	tyLyrC0008MsgBox : 	STRUCT
		tyBitmapIcon : tyUIBitmap;
		tyTxtTitle : tyUITxt;
		tyTxtMsg : tyUITxt;
		tyBtnYes : tyUIBtn;
		tyBtnNo : tyUIBtn;
		tyLyr : tyUILyr;
	END_STRUCT;
	tyLyrC0009Info : 	STRUCT
		tyStringInfo : tyUILString;
		tyHotspotClose : tyUIHotspot;
		tyLyr : tyUILyr;
	END_STRUCT;
	tyLyrC0010RcyMsg : 	STRUCT
		tyHotspotClose : tyUIHotspot;
		tyLyr : tyUILyr;
		tyTxtMsg : tyUIAlmTxt;
	END_STRUCT;
	tyLyrC0011Loading : 	STRUCT
		tyUILoad : tyUIBitmap;
		tyStringMsg : tyUILString;
		tyLyr : tyUILyr;
	END_STRUCT;
	tyLyrC0012RcpPopUp : 	STRUCT
		tyStringInfo : tyUILString;
		tyHotspotClose : tyUIHotspot;
		tyLyr : tyUILyr;
	END_STRUCT;
END_TYPE

(**)
(*Layer*)

TYPE
	tyLyrP0000SSaver : 	STRUCT
		tyTxtMcStat : tyUITxt;
		tyTxtMcNm : tyUILString;
		tyBitmapStat : tyUIBitmap;
		tyLyr : tyUILyr;
	END_STRUCT;
END_TYPE

(**)

TYPE
	tyLyrP0001Startup : 	STRUCT
		tyBarGraphStartup : tyUIBarGraph;
		tyTxtStartupStat : tyUITxt;
		tyLyr : tyUILyr;
	END_STRUCT;
	tyLyrP0001Initial : 	STRUCT
		tyLyr : tyUILyr;
	END_STRUCT;
END_TYPE

(**)

TYPE
	tyLyrP0002Menu : 	STRUCT
		tyBtnAlm : tyUIBtn;
		tyBtnCommCtrl : tyUIBtn;
		tyBtnGenInput : tyUIBtn;
		tyBtnGenOutput : tyUIBtn;
		tyBtnLang : tyUIBtn;
		tyBtnLFCtrl : tyUIBtn;
		tyBtnLFSet : tyUIBtn;
		tyBtnLogin : tyUIBtn;
		tyBtnMcInfo : tyUIBtn;
		tyBtnMcSet : tyUIBtn;
		tyBtnMnlRst : tyUIBtn;
		tyBtnMovCtrl : tyUIBtn;
		tyBtnOpt : tyUIBtn;
		tyBtnProdSel : tyUIBtn;
		tyBtnProdSet : tyUIBtn;
		tyBtnSimu : tyUIBtn;
		tyBtnUsrMgmt : tyUIBtn;
		tyBitmapMaskProdSetLCS : tyUIBitmap;
		tyGenMaskLyr : tyUILyr;
		tySetMaskLyr : tyUILyr;
		tyHotspotRstRtnBrd : tyUIHotspot;
	END_STRUCT;
END_TYPE

(**)

TYPE
	tyLyrP0100Login : 	STRUCT
		tyBtnLogin : tyUIBtn;
		tyHotspotShowLoginLvl : tyUIHotspot;
		tyHotspotBypassLogin : tyUIHotspot;
		tyStringPw : tyUIString;
		tyStringUsrNm : tyUIString;
		tyLyr : tyUILyr;
	END_STRUCT;
	tyLyrP0100Logout : 	STRUCT
		tyBtnLogout : tyUIBtn;
		tyLyr : tyUILyr;
	END_STRUCT;
END_TYPE

(**)

TYPE
	tyLyrP0200OpsGen : 	STRUCT
		a_tyHotspotRcyMsg : ARRAY[1..c_uiP0200TableSize]OF tyUIHotspot;
		a_tyStringAlm : ARRAY[1..c_uiP0200TableSize]OF tyUILString;
		tyBitmapDSCommIcon : tyUIBitmap;
		tyBitmapDSCommIn : tyUIBitmap;
		tyBitmapDSCommOut : tyUIBitmap;
		tyBitmapDSCommIn1 : tyUIBitmap;
		tyBitmapDSCommOut1 : tyUIBitmap;
		tyBitmapUSCommIcon : tyUIBitmap;
		tyBitmapUSCommIn : tyUIBitmap;
		tyBitmapUSCommOut : tyUIBitmap;
		tyBitmapUSCommIn1 : tyUIBitmap;
		tyBitmapUSCommOut1 : tyUIBitmap;
		tyBitmapUSCommIcon2 : tyUIBitmap;
		tyBitmapUSCommIn2 : tyUIBitmap;
		tyBitmapUSCommOut2 : tyUIBitmap;
		tyBitmapDir1 : tyUIBitmap;
		tyBitmapDir2 : tyUIBitmap;
		tyBitmapConvPCB : tyUIBitmap;
		tyBitmapStackerPCB : tyUIBitmap;
		tyBitmapAccDat : tyUIBitmap;
		tyBitmapRlsNewProd : tyUIBitmap;
		tyBitmapMc : tyUIBitmap;
		tyBitmapBypassTopCover1 : tyUIBitmap;
		tyBtnBypassTopCover1 : tyUIBtn;
		tyBtnAccDat : tyUIBtn;
		tyBtnRlsNewProd : tyUIBtn;
		tyBtnPCBReset : tyUIBtn;
		tyHotspotMc : tyUIHotspot;
		tyHotspotDSVirtual : tyUIHotspot;
		tyHotspotUSVirtual : tyUIHotspot;
		tyHotspotDSVirtual1 : tyUIHotspot;
		tyHotspotUSVirtual1 : tyUIHotspot;
		tyHotspotUSVirtual2 : tyUIHotspot;
		tyTxtUS : tyUITxt;
		tyTxtUS1 : tyUITxt;
		tyTxtUS2 : tyUITxt;
		tyTxtDS : tyUITxt;
		tyTxtDS1 : tyUITxt;
		tyTxtLdrInActiveCtrl : tyUITxt;
		tyBitmapWarningLF : tyUIBitmap;
		tyLyr : tyUILyr;
	END_STRUCT;
	tyLyrP0200OpsUSVSMEMA : 	STRUCT
		tyBtnUBAStat : tyUIBtn;
		tyBtnUBA : tyUIBtn;
		tyBtnDual : tyUIBtn;
		tyLyr : tyUILyr;
	END_STRUCT;
	tyLyrP0200OpsDSVSMEMA : 	STRUCT
		tyBtnDSBStat : tyUIBtn;
		tyBtnDSB : tyUIBtn;
		tyBtnDual : tyUIBtn;
		tyLyr : tyUILyr;
	END_STRUCT;
	tyLyrP0200OpsUSVSMEMA1 : 	STRUCT
		tyBtnUBAStat : tyUIBtn;
		tyBtnUBA : tyUIBtn;
		tyBtnDual : tyUIBtn;
		tyLyr : tyUILyr;
	END_STRUCT;
	tyLyrP0200OpsDSVSMEMA1 : 	STRUCT
		tyBtnDSBStat : tyUIBtn;
		tyBtnDSB : tyUIBtn;
		tyBtnDual : tyUIBtn;
		tyLyr : tyUILyr;
	END_STRUCT;
	tyLyrP0200OpsUSVSMEMA2 : 	STRUCT
		tyBtnUBAStat : tyUIBtn;
		tyBtnUBA : tyUIBtn;
		tyBtnDual : tyUIBtn;
		tyLyr : tyUILyr;
	END_STRUCT;
	tyLyrP0200OpsBypsInitConv : 	STRUCT
		tyBtnBypsInitConv : tyUIBtn;
		tyHotspotClose : tyUIHotspot;
		tyLyr : tyUILyr;
	END_STRUCT;
END_TYPE

(**)

TYPE
	tyLyrP0201OpsConv : 	STRUCT
		tyBitmapAccDat : tyUIBitmap;
		tyBitmapRlsNewProd : tyUIBitmap;
		tyBitmapConvPCB : tyUIBitmap;
		tyBitmapBypassTopCover1 : tyUIBitmap;
		tyBtnAccDat : tyUIBtn;
		tyBtnRlsNewProd : tyUIBtn;
		tyBtnChgParam : tyUIBtn;
		tyBtnBypassTopCover1 : tyUIBtn;
		tyHotspotIOMonitor : tyUIHotspot;
		tyNumProdWidth : tyUINum;
		tyNumProdWidth2 : tyUINum;
		tyStringProdNm : tyUILString;
		tyStringMcStatus : tyUILString;
		tyTxtMod : tyUITxt;
		tyLblFlippedBrd : tyUITxt;
		tyTxtFlippedBrd : tyUITxt;
		tyStringMatchCode : tyUIString;
		tyTxtLdrInActiveCtrl : tyUITxt;
		tyBitmapWarningLF : tyUIBitmap;
		tyBitmapMc : tyUIBitmap;
		tyLyr : tyUILyr;
		tyHotspotShowLRcp : tyUIHotspot;
	END_STRUCT;
	tyLyrP0201OpsConvIOMonitor : 	STRUCT
		tyBtnSafetyRlySig : tyUIBtn;
		tyBtnEStop : tyUIBtn;
		tyBtnCoverSWSig : tyUIBtn;
		tyBtnUBA : tyUIBtn;
		tyBtnUBAStat : tyUIBtn;
		tyBtnDSB : tyUIBtn;
		tyBtnConvLftSen : tyUIBtn;
		tyBtnConvRgtSen : tyUIBtn;
		tyBtnPressureSW : tyUIBtn;
		tyBtnThermalPrtSig : tyUIBtn;
		tyBtnCoatingSen : tyUIBtn;
		tyBtnUSWidthChkSen : tyUIBtn;
		tyBtnDSWidthChkSen : tyUIBtn;
		tyBtnInvertHomeSen : tyUIBtn;
		tyBtnInvertRemoteSen : tyUIBtn;
		tyBtnInletShutterOpenRS : tyUIBtn;
		tyBtnInletShutterCloseRS : tyUIBtn;
		tyBtnOutletShutterOpenRS : tyUIBtn;
		tyBtnOutletShutterCloseRS : tyUIBtn;
		tyBtnSafetyRlyRst : tyUIBtn;
		tyBtnTLGreen : tyUIBtn;
		tyBtnTLAmber : tyUIBtn;
		tyBtnTLRed : tyUIBtn;
		tyBtnTLWhite : tyUIBtn;
		tyBtnTLBlue : tyUIBtn;
		tyBtnBuzzer : tyUIBtn;
		tyBtnCoatingRetCtrl : tyUIBtn;
		tyBtnUSB : tyUIBtn;
		tyBtnDBA : tyUIBtn;
		tyBtnDBAStat : tyUIBtn;
		tyBtnConvMtrCW : tyUIBtn;
		tyBtnConvMtrCCW : tyUIBtn;
		tyBtnStprUnblkCtrl : tyUIBtn;
		tyBtnStprBlkCtrl : tyUIBtn;
		tyBtnInvertHome : tyUIBtn;
		tyBtnInvertRemote : tyUIBtn;
		tyBtnInvertBrake : tyUIBtn;
		tyBtnMtrPwrRly : tyUIBtn;
		tyBtnClampCtrl : tyUIBtn;
		tyBtnUnclampCtrl : tyUIBtn;
		tyBtnInShutterOpenCtrl : tyUIBtn;
		tyBtnInShutterCloseCtrl : tyUIBtn;
		tyBtnOutShutterOpenCtrl : tyUIBtn;
		tyBtnOutShutterCloseCtrl : tyUIBtn;
		tyHotspotClose : tyUIHotspot;
		tyLyr : tyUILyr;
	END_STRUCT;
	tyLyrP0201OpsConvIOMonitorMSafe : 	STRUCT
		tyBtnSafetyRlySig : tyUIBtn;
		tyBtnEStop : tyUIBtn;
		tyBtnCoverSWSig : tyUIBtn;
		tyBtnUBA : tyUIBtn;
		tyBtnUBAStat : tyUIBtn;
		tyBtnDSB : tyUIBtn;
		tyBtnConvLftSen : tyUIBtn;
		tyBtnConvRgtSen : tyUIBtn;
		tyBtnPressureSW : tyUIBtn;
		tyBtnThermalPrtSig : tyUIBtn;
		tyBtnCoatingSen : tyUIBtn;
		tyBtnUSWidthChkSen : tyUIBtn;
		tyBtnDSWidthChkSen : tyUIBtn;
		tyBtnInvertHomeSen : tyUIBtn;
		tyBtnInvertRemoteSen : tyUIBtn;
		tyBtnInletShutterOpenRS : tyUIBtn;
		tyBtnInletShutterCloseRS : tyUIBtn;
		tyBtnOutletShutterOpenRS : tyUIBtn;
		tyBtnOutletShutterCloseRS : tyUIBtn;
		tyBtnClamp2Sen : tyUIBtn;
		tyBtnClamp3Sen : tyUIBtn;
		tyBtnClampRS1 : tyUIBtn;
		tyBtnUnClampRS1 : tyUIBtn;
		tyBtnClampRS2 : tyUIBtn;
		tyBtnUnClampRS2 : tyUIBtn;
		tyBtnClampRS3 : tyUIBtn;
		tyBtnUnClampRS3 : tyUIBtn;
		tyBtnCoverSWSig2 : tyUIBtn;
		tyBtnSafetySigFromUS : tyUIBtn;
		tyBtnSafetySigFromDS : tyUIBtn;
		tyBtnUnlockCoverSigFromUS : tyUIBtn;
		tyBtnUnlockCoverSigFromDS : tyUIBtn;
		tyBtnCoverUnlockPB1 : tyUIBtn;
		tyBtnSafetyRlyRst : tyUIBtn;
		tyBtnTLGreen : tyUIBtn;
		tyBtnTLAmber : tyUIBtn;
		tyBtnTLRed : tyUIBtn;
		tyBtnTLWhite : tyUIBtn;
		tyBtnTLBlue : tyUIBtn;
		tyBtnBuzzer : tyUIBtn;
		tyBtnCoatingRetCtrl : tyUIBtn;
		tyBtnUSB : tyUIBtn;
		tyBtnDBA : tyUIBtn;
		tyBtnDBAStat : tyUIBtn;
		tyBtnConvMtrCW : tyUIBtn;
		tyBtnConvMtrCCW : tyUIBtn;
		tyBtnInvertHome : tyUIBtn;
		tyBtnInvertRemote : tyUIBtn;
		tyBtnInvertBrake : tyUIBtn;
		tyBtnMtrPwrRly : tyUIBtn;
		tyBtnInShutterOpenCtrl : tyUIBtn;
		tyBtnInShutterCloseCtrl : tyUIBtn;
		tyBtnOutShutterOpenCtrl : tyUIBtn;
		tyBtnOutShutterCloseCtrl : tyUIBtn;
		tyBtnClamp1Ctrl : tyUIBtn;
		tyBtnUnclamp1Ctrl : tyUIBtn;
		tyBtnClamp2Ctrl : tyUIBtn;
		tyBtnUnclamp2Ctrl : tyUIBtn;
		tyBtnClamp3Ctrl : tyUIBtn;
		tyBtnUnclamp3Ctrl : tyUIBtn;
		tyBtnTopCvrUnlckToDS : tyUIBtn;
		tyBtnTopCvrUnlckToUS : tyUIBtn;
		tyBtniMachineSafetySigToDS : tyUIBtn;
		tyBtnMachineSafetySigToUS : tyUIBtn;
		tyBtnPBLED1 : tyUIBtn;
		tyBtnBypassTopCover1 : tyUIBtn;
		tyBtnSafetyTopCoverSWCoil1 : tyUIBtn;
		tyHotspotClose : tyUIHotspot;
		tyLyr : tyUILyr;
	END_STRUCT;
	tyLyrP0201OpsConvIOMonitorXStd : 	STRUCT
		tyBtnSafetyRlySig : tyUIBtn;
		tyBtnEStop : tyUIBtn;
		tyBtnCoverSWSig : tyUIBtn;
		tyBtnUBA : tyUIBtn;
		tyBtnUBAStat : tyUIBtn;
		tyBtnDSB : tyUIBtn;
		tyBtnUBA2 : tyUIBtn;
		tyBtnUBAStat2 : tyUIBtn;
		tyBtnConvLftSen : tyUIBtn;
		tyBtnConvRgtSen : tyUIBtn;
		tyBtnPressureSW : tyUIBtn;
		tyBtnThermalPrtSig : tyUIBtn;
		tyBtnCoatingSen : tyUIBtn;
		tyBtnUSWidthChkSen : tyUIBtn;
		tyBtnDSWidthChkSen : tyUIBtn;
		tyBtnInvertHomeSen : tyUIBtn;
		tyBtnInvertRemoteSen : tyUIBtn;
		tyBtnInletShutterOpenRS : tyUIBtn;
		tyBtnInletShutterCloseRS : tyUIBtn;
		tyBtnOutletShutterOpenRS : tyUIBtn;
		tyBtnOutletShutterCloseRS : tyUIBtn;
		tyBtnClamp2Sen : tyUIBtn;
		tyBtnClamp3Sen : tyUIBtn;
		tyBtnClampRS1 : tyUIBtn;
		tyBtnUnClampRS1 : tyUIBtn;
		tyBtnClampRS2 : tyUIBtn;
		tyBtnUnClampRS2 : tyUIBtn;
		tyBtnClampRS3 : tyUIBtn;
		tyBtnUnClampRS3 : tyUIBtn;
		tyBtnSafetyRlyRst : tyUIBtn;
		tyBtnTLGreen : tyUIBtn;
		tyBtnTLAmber : tyUIBtn;
		tyBtnTLRed : tyUIBtn;
		tyBtnTLWhite : tyUIBtn;
		tyBtnTLBlue : tyUIBtn;
		tyBtnBuzzer : tyUIBtn;
		tyBtnCoatingRetCtrl : tyUIBtn;
		tyBtnUSB : tyUIBtn;
		tyBtnDBA : tyUIBtn;
		tyBtnDBAStat : tyUIBtn;
		tyBtnUSB2 : tyUIBtn;
		tyBtnConvMtrCW : tyUIBtn;
		tyBtnConvMtrCCW : tyUIBtn;
		tyBtnInvertHome : tyUIBtn;
		tyBtnInvertRemote : tyUIBtn;
		tyBtnInvertBrake : tyUIBtn;
		tyBtnMtrPwrRly : tyUIBtn;
		tyBtnInShutterOpenCtrl : tyUIBtn;
		tyBtnInShutterCloseCtrl : tyUIBtn;
		tyBtnOutShutterOpenCtrl : tyUIBtn;
		tyBtnOutShutterCloseCtrl : tyUIBtn;
		tyBtnClamp1Ctrl : tyUIBtn;
		tyBtnUnclamp1Ctrl : tyUIBtn;
		tyBtnClamp2Ctrl : tyUIBtn;
		tyBtnUnclamp2Ctrl : tyUIBtn;
		tyBtnClamp3Ctrl : tyUIBtn;
		tyBtnUnclamp3Ctrl : tyUIBtn;
		tyHotspotClose : tyUIHotspot;
		tyLyr : tyUILyr;
	END_STRUCT;
	tyLyrP0201OpsConvChgParam : 	STRUCT
		tyDrpDnMcMode : tyUIDrpDn;
		tyDrpDnFlippedBrd : tyUIDrpDn;
		tyNumProdWidth : tyUINum;
		tyBtnSave : tyUIBtn;
		tyBtnCancel : tyUIBtn;
		tyLyr : tyUILyr;
	END_STRUCT;
	tyLyrP0201OpsConvBypsInitConv : 	STRUCT
		tyBtnBypsInitConv : tyUIBtn;
		tyHotspotClose : tyUIHotspot;
		tyLyr : tyUILyr;
	END_STRUCT;
END_TYPE

(**)

TYPE
	tyLyrP0300McInfo : 	STRUCT
		tyTxtNtAddr : tyUITxt;
		tyStringMcNm : tyUIString;
		tyStringJobNo : tyUIString;
		tyStringSoftwareVer : tyUIString;
		tyBtnPlaySong : tyUIBtn;
		tyDrpDnSong : tyUIDrpDn;
		tyLyr : tyUILyr;
	END_STRUCT;
END_TYPE

(**)

TYPE
	tyLyrP0400ProdSel : 	STRUCT
		tyBtnLoad : tyUIBtn;
		tyBtnPreview : tyUIBtn;
		tyNumProdWidth : tyUINum;
		tyNumProdWidth2 : tyUINum;
		tyStringRecipeNm : tyUILString;
		tyStringSearch : tyUILString;
		tyTableRecipe : tyUITable;
		tyTxtMcMod : tyUITxt;
		tyTxtFlippedBrd : tyUITxt;
		tyTxtMatchCodeLbl : tyUITxt;
		tyStringMatchCode : tyUIString;
		tyBtnSort : tyUIBtn;
		tyLyr : tyUILyr;
		tyHotspotShowLRcp : tyUIHotspot;
	END_STRUCT;
	tyLyrP0400RcpDet : 	STRUCT
		tyHotspotClose : tyUIHotspot;
		tyNumProdWidth : tyUINum;
		tyNumProdWidth2 : tyUINum;
		tyStringRecipeNm : tyUILString;
		tyTxtMcMod : tyUITxt;
		tyTxtFlippedBrd : tyUITxt;
		tyTxtMatchCodeLbl : tyUITxt;
		tyStringMatchCode : tyUIString;
		tyLyr : tyUILyr;
		tyHotspotShowLRcp : tyUIHotspot;
	END_STRUCT;
END_TYPE

(**)

TYPE
	tyLyrP0600Alm : 	STRUCT
		tyBtnHistory : tyUIBtn;
		tyBtnCurr : tyUIBtn;
		a_tyStringAlm : ARRAY[0..c_uiP0600TableSize]OF tyUILString;
		a_tyHotspotAlm : ARRAY[0..c_uiP0600TableSize]OF tyUIHotspot;
		tyLyr : tyUILyr;
		tyAlarm : tyUIAlarm;
		tyBtnHistoryUp : tyUIBtn;
		tyBtnHistoryDown : tyUIBtn;
	END_STRUCT;
END_TYPE

(**)

TYPE
	tyLyrP0700LFCtrl : 	STRUCT
		tyBtnChgAll : tyUIBtn;
		tyBtnChgSeqAuto : tyUIBtn := (uiMaskRtStat:=0);
		tyBtnChgSeqMnl : tyUIBtn := (uiMaskRtStat:=0);
		tyBtnSyncTm : tyUIBtn;
		tyBitmapChgAll : tyUIBitmap;
		tyBitmapChgSeqAuto : tyUIBitmap;
		tyBitmapChgSeqMnl : tyUIBitmap;
		tyBitmapSyncTm : tyUIBitmap;
		tyTable1List : tyUITable1;
		tyLyr : tyUILyr;
	END_STRUCT;
END_TYPE

(**)

TYPE
	tyLyrP0900GenIn : 	STRUCT
		tyBtnEStop : tyUIBtn;
		tyBtnCoverSW : tyUIBtn;
		tyBtnSafety : tyUIBtn;
		tyLyr : tyUILyr;
		tyBtnUSWidthChkSen : tyUIBtn;
		tyBtnDSWidthChkSen : tyUIBtn;
		tyBtnPressureSW : tyUIBtn;
		tyBtnThermalPrtSig : tyUIBtn;
		tyBtnUnlkCovPB : tyUIBtn;
		tyBtnSafetySigFromUS : tyUIBtn;
		tyBtnSafetySigFromDS : tyUIBtn;
		tyBtnUlkCoverFromDS : tyUIBtn;
		tyBtnUlkCoverFromUS : tyUIBtn;
		tyBtnTopCovSwSIg : tyUIBtn;
		tySigLyr : tyUILyr;
		tyWidthChkLyr : tyUILyr;
		tyMachSafetyLyr : tyUILyr;
	END_STRUCT;
END_TYPE

(**)

TYPE
	tyLyrP0910GenOut : 	STRUCT
		tyBtnTLGreen : tyUIBtn;
		tyBtnTLAmber : tyUIBtn;
		tyBtnTLRed : tyUIBtn;
		tyBtnTLRed1 : tyUIBtn;
		tyBtnTLBlue : tyUIBtn;
		tyBtnTLWhite : tyUIBtn;
		tyBtnBuzzer : tyUIBtn;
		tyBtnSafety : tyUIBtn;
		tyBtnUlkCovPBLED : tyUIBtn;
		tyBtnUlkCovHoldRely : tyUIBtn;
		tyBtnSftUlkCovSWCoil : tyUIBtn;
		tyBtnTopCovUlkUSDS : tyUIBtn;
		tyBtnSftSigToUSDS : tyUIBtn;
		tyUlkCovLyr : tyUILyr;
		tyMacSafetyLyr : tyUILyr;
		tyLyr : tyUILyr;
		tyTLLyr : tyUILyr;
	END_STRUCT;
END_TYPE

(**)

TYPE
	tyLyrP0920MtrNPneuCtrl : 	STRUCT
		tyBtnAW : tyUIBtn;
		tyBitmapAW : tyUIBitmap;
		tyBtnShutter : tyUIBtn;
		tyBitmapShutter : tyUIBitmap;
		tyBtnClampNoRS : tyUIBtn;
		tyBtnClampWithRS : tyUIBtn;
		tyBtnStopper : tyUIBtn;
		tyBtnConv : tyUIBtn;
		tyBitmapConv : tyUIBitmap;
		tyLyr : tyUILyr;
	END_STRUCT;
END_TYPE

(**)

TYPE
	tyLyrP0921ClampNoRSCom : 	STRUCT
		tyBitmapMc : tyUIBitmap;
		tyBtnDCCtrl : tyUIBtn;
		tyBtnExtRS : tyUIBtn;
		tyBtnRetRS : tyUIBtn;
		tyTxtSubTitle : tyUITxt;
		tyLyr : tyUILyr;
	END_STRUCT;
	tyLyrP0921ClampNoRSDC : 	STRUCT
		tyBtnExt : tyUIBtn;
		tyBtnRet : tyUIBtn;
		tyLyr : tyUILyr;
	END_STRUCT;
	tyLyrP0921ClampNoRSFB : 	STRUCT
		tyStringStat : tyUILString;
		tyBtnExt : tyUIBtn;
		tyBtnRet : tyUIBtn;
		tyLyr : tyUILyr;
	END_STRUCT;
END_TYPE

(**)

TYPE
	tyLyrP0922InletShutterCom : 	STRUCT
		tyBtnSwitch : tyUIBtn;
		tyBitmapMc : tyUIBitmap;
		tyBtnOpenRS : tyUIBtn;
		tyBtnCloseRS : tyUIBtn;
		tyLyr : tyUILyr;
	END_STRUCT;
	tyLyrP0922InletShutterDC : 	STRUCT
		tyBtnOpen : tyUIBtn;
		tyBtnClose : tyUIBtn;
		tyLyr : tyUILyr;
	END_STRUCT;
	tyLyrP0922InletShutterFB : 	STRUCT
		tyStringStat : tyUILString;
		tyBtnOpen : tyUIBtn;
		tyBtnClose : tyUIBtn;
		tyLyr : tyUILyr;
	END_STRUCT;
	tyLyrP0922InletShutterDis : 	STRUCT
		tyLyr : tyUILyr;
	END_STRUCT;
	tyLyrP0922OutletShutterCom : 	STRUCT
		tyBtnSwitch : tyUIBtn;
		tyBitmapMc : tyUIBitmap;
		tyBtnOpenRS : tyUIBtn;
		tyBtnCloseRS : tyUIBtn;
		tyLyr : tyUILyr;
	END_STRUCT;
	tyLyrP0922OutletShutterDC : 	STRUCT
		tyBtnOpen : tyUIBtn;
		tyBtnClose : tyUIBtn;
		tyLyr : tyUILyr;
	END_STRUCT;
	tyLyrP0922OutletShutterFB : 	STRUCT
		tyStringStat : tyUILString;
		tyBtnOpen : tyUIBtn;
		tyBtnClose : tyUIBtn;
		tyLyr : tyUILyr;
	END_STRUCT;
	tyLyrP0922OutletShutterDis : 	STRUCT
		tyLyr : tyUILyr;
	END_STRUCT;
END_TYPE

(**)

TYPE
	tyLyrP0923StopperCom : 	STRUCT
		tyBtnDCCtrl : tyUIBtn;
		tyBitmapMc : tyUIBitmap;
		tyLyr : tyUILyr;
	END_STRUCT;
	tyLyrP0923StopperDC : 	STRUCT
		tyBtnExtend : tyUIBtn;
		tyBtnRetract : tyUIBtn;
		tyLyr : tyUILyr;
	END_STRUCT;
	tyLyrP0923StopperFB : 	STRUCT
		tyBtnExtend : tyUIBtn;
		tyBtnRetract : tyUIBtn;
		tyStringStat : tyUILString;
		tyLyr : tyUILyr;
	END_STRUCT;
END_TYPE

(**)

TYPE
	tyLyrP0924Clamp1WithRSCom : 	STRUCT
		tyBtnSwitch : tyUIBtn;
		tyBitmapMc : tyUIBitmap;
		tyBtnClampRS : tyUIBtn;
		tyBtnUnClampRS : tyUIBtn;
		tyLyr : tyUILyr;
	END_STRUCT;
	tyLyrP0924Clamp1WithRSDC : 	STRUCT
		tyBtnExt : tyUIBtn;
		tyBtnRet : tyUIBtn;
		tyLyr : tyUILyr;
	END_STRUCT;
	tyLyrP0924Clamp1WithRSDis : 	STRUCT
		tyLyr : tyUILyr;
	END_STRUCT;
	tyLyrP0924Clamp1WithRSFB : 	STRUCT
		tyStringStat : tyUILString;
		tyBtnExt : tyUIBtn;
		tyBtnRet : tyUIBtn;
		tyLyr : tyUILyr;
	END_STRUCT;
	tyLyrP0924Clamp2WithRSCom : 	STRUCT
		tyBtnSwitch : tyUIBtn;
		tyBitmapMc : tyUIBitmap;
		tyBtnClampRS : tyUIBtn;
		tyBtnUnClampRS : tyUIBtn;
		tyLyr : tyUILyr;
	END_STRUCT;
	tyLyrP0924Clamp2WithRSDC : 	STRUCT
		tyBtnExt : tyUIBtn;
		tyBtnRet : tyUIBtn;
		tyLyr : tyUILyr;
	END_STRUCT;
	tyLyrP0924Clamp2WithRSDis : 	STRUCT
		tyLyr : tyUILyr;
	END_STRUCT;
	tyLyrP0924Clamp2WithRSFB : 	STRUCT
		tyStringStat : tyUILString;
		tyBtnExt : tyUIBtn;
		tyBtnRet : tyUIBtn;
		tyLyr : tyUILyr;
	END_STRUCT;
	tyLyrP0924Clamp3WithRSCom : 	STRUCT
		tyBtnSwitch : tyUIBtn;
		tyBitmapMc : tyUIBitmap;
		tyBtnClampRS : tyUIBtn;
		tyBtnUnClampRS : tyUIBtn;
		tyLyr : tyUILyr;
	END_STRUCT;
	tyLyrP0924Clamp3WithRSDC : 	STRUCT
		tyBtnExt : tyUIBtn;
		tyBtnRet : tyUIBtn;
		tyLyr : tyUILyr;
	END_STRUCT;
	tyLyrP0924Clamp3WithRSDis : 	STRUCT
		tyLyr : tyUILyr;
	END_STRUCT;
	tyLyrP0924Clamp3WithRSFB : 	STRUCT
		tyStringStat : tyUILString;
		tyBtnExt : tyUIBtn;
		tyBtnRet : tyUIBtn;
		tyLyr : tyUILyr;
	END_STRUCT;
END_TYPE

(**)

TYPE
	tyLyrP0931ConvCom : 	STRUCT
		tyBtnLft : tyUIBtn;
		tyBtnRgt : tyUIBtn;
		tyBitmapMc : tyUIBitmap;
		tyBtnDCCtrl : tyUIBtn;
	END_STRUCT;
	tyLyrP0931ConvDC : 	STRUCT
		tyBtnConvLToR : tyUIBtn;
		tyBtnConvRToL : tyUIBtn;
		tyBtnStop : tyUIBtn := (bRtLk:=TRUE,bValue:=TRUE);
		tyLyr : tyUILyr := (uiRtStat:=1);
	END_STRUCT;
	tyLyrP0931ConvFB : 	STRUCT
		tyBtnEnt : tyUIBtn;
		tyBtnExit : tyUIBtn;
		tyBtnPreExit : tyUIBtn;
		tyBtnStop : tyUIBtn := (bRtLk:=TRUE,bValue:=TRUE);
		tyLyr : tyUILyr;
		tyStringStat : tyUILString;
	END_STRUCT;
	tyLyrP0931InvCom : 	STRUCT
		tyBtnHomeSen : tyUIBtn;
		tyBtnRemoteSen : tyUIBtn;
		tyBtnDCCtrl : tyUIBtn;
		tyBitmapMc : tyUIBitmap;
	END_STRUCT;
	tyLyrP0931InvDC : 	STRUCT
		tyBtnBrake : tyUIBtn;
		tyBtnCCW : tyUIBtn;
		tyBtnCW : tyUIBtn;
		tyLyr : tyUILyr := (uiRtStat:=1);
	END_STRUCT;
	tyLyrP0931InvFB : 	STRUCT
		tyBtnCCW : tyUIBtn;
		tyBtnCW : tyUIBtn;
		tyBtnStop : tyUIBtn := (bRtLk:=TRUE,bValue:=TRUE);
		tyLyr : tyUILyr;
		tyStringStat : tyUILString;
	END_STRUCT;
END_TYPE

(**)

TYPE
	tyLyrP0934AW : 	STRUCT
		tyBitmapMc : tyUIBitmap;
		tyBtnGo : tyUIBtn;
		tyNumNewWidth : tyUINum;
		tyLyr : tyUILyr;
	END_STRUCT;
END_TYPE

(**)
(**)

TYPE
	tyLyrP0940CommCtrlDSSMEMA : 	STRUCT
		tyBtnDBA : tyUIBtn;
		tyBtnDBAStat : tyUIBtn;
		tyBtnDSB : tyUIBtn;
		tyLyr : tyUILyr;
	END_STRUCT;
	tyLyrP0940CommCtrlUSSMEMA : 	STRUCT
		tyBtnUBA : tyUIBtn;
		tyBtnUBAStat : tyUIBtn;
		tyBtnUSB : tyUIBtn;
		tyLyr : tyUILyr;
	END_STRUCT;
	tyLyrP0940CommCtrlUSSMEMA2 : 	STRUCT
		tyBtnUBA : tyUIBtn;
		tyBtnUBAStat : tyUIBtn;
		tyBtnUSB : tyUIBtn;
		tyLyr : tyUILyr;
	END_STRUCT;
END_TYPE

(**)

TYPE
	tyLyrP0950Simu : 	STRUCT
		tyBtnSimu : tyUIBtn := (bRtLk:=TRUE,bValue:=TRUE);
		tyBtnStart : tyUIBtn;
		tyBtnStop : tyUIBtn;
		tyLyr : tyUILyr;
	END_STRUCT;
END_TYPE

(**)

TYPE
	tyLyrP1000Lang : 	STRUCT
		tyBtnChinese : tyUIBtn;
		tyBtnEnglish : tyUIBtn;
		tyBtnGerman : tyUIBtn;
		tyNumYear : tyUINum;
		tyNumMonth : tyUINum;
		tyNumDay : tyUINum;
		tyNumHour : tyUINum;
		tyNumMinute : tyUINum;
		tyNumSecond : tyUINum;
		tyLyr : tyUILyr;
	END_STRUCT;
END_TYPE

(**)

TYPE
	tyLyrP1020McSetNavi : 	STRUCT
		tyBtnMcSet : tyUIBtn;
		tyBtnVCommSet : tyUIBtn;
		tyBtnHCommSet : tyUIBtn;
		tyBtnAntiGapSet : tyUIBtn;
		tyLyr : tyUILyr;
	END_STRUCT;
END_TYPE

(**)

TYPE
	tyLyrP1021McSetGen : 	STRUCT
		tyBtnAutoStepEn : tyUIBtn;
		tyBtnAWDis : tyUIBtn;
		tyBtnChgParamEn : tyUIBtn;
		tyBtnHermesRmtEn : tyUIBtn;
		tyBtnMnlAccDat : tyUIBtn;
		tyBtnVSMEMAEn : tyUIBtn;
		tyDrpDnDefaultMcMod : tyUIDrpDn;
		tyDrpDnDefaultFlippedBrd : tyUIDrpDn;
		tyDrpDnNetworkMod : tyUIDrpDn;
		tyTxtLblFlippedBrd : tyUITxt;
		tyHermesRemoteEn : tyUIBtn;
		tyLyrGen1 : tyUILyr;
		tyLyrGen2 : tyUILyr;
		tyNumConvInitTm : tyUINum;
		tyNumTranInErrDlyTm : tyUINum;
		tyNumTranOutErrDlyTm : tyUINum;
		tyNumWidthAtHm : tyUINum;
		tyTxtWidthOffset : tyUITxt;
		tyNumWidthOffset : tyUINum;
		tyStringMcNm : tyUIString;
		tyTxtWidthAtHm : tyUITxt;
		tyBtnSSaverEn : tyUIBtn;
		tyNumSSaverTm : tyUINum;
		tyTxtSSaverTm : tyUITxt;
		tyStringSubnetMask : tyUIString;
		tyStringIPAddr : tyUIString;
		tyNumStopperAtLftPos : tyUINum;
		tyNumStopperAtRgtPos : tyUINum;
		tyBtnStopperAtLftPosTeach : tyUIBtn;
		tyBtnStopperAtRgtPosTeach : tyUIBtn;
		tyBtnClampDis : tyUIBtn;
		tyBtnStopperDis : tyUIBtn;
		tyNumAutoLogoutTm : tyUINum;
		tyTxtLblAutoLogoutTm : tyUITxt;
		tyBtnAutoLogoutEn : tyUIBtn;
		tyBtnLFBuzMute : tyUIBtn;
	END_STRUCT;
	tyLyrP1021McSetNetwork : 	STRUCT
		tyStringIPAddr : tyUIString;
		tyStringSubnetMask : tyUIString;
		tyBtnSave : tyUIBtn;
		tyBtnCancel : tyUIBtn;
		tyLyr : tyUILyr;
	END_STRUCT;
END_TYPE

(**)

TYPE
	tyLyrP1022McSetVCommSel : 	STRUCT
		tyBtnLF : tyUIBtn;
		tyBtnLCSLF : tyUIBtn;
		tyBtnLCSReqRcp : tyUIBtn;
		tyBtnLCSManageRcp : tyUIBtn;
		tyBtnLCSLiveDat : tyUIBtn;
		tyLyr : tyUILyr;
	END_STRUCT;
	tyLyrP1022McSetVCommLF : 	STRUCT
		tyBtnLeaderMc : tyUIBtn;
		tyBtnSectionLdr : tyUIBtn;
		tyBtnDBAOnWOAlign : tyUIBtn;
		tyBtnUSWidthChkEn : tyUIBtn;
		tyBtnDSWidthChkEn : tyUIBtn;
		tyBtnSeqStayActive : tyUIBtn;
		tyLyr : tyUILyr;
	END_STRUCT;
	tyLyrP1022McSetVCommSvy : 	STRUCT
		tyNumSndAliveTm : tyUINum;
		tyNumSvySystemPort : tyUINum;
		tyBtnConfiguration : tyUIBtn;
		tyBtnCheckAliveResponse : tyUIBtn;
		tyBtnBoardTracking : tyUIBtn;
		tyBtnQueryWorkOrderInfo : tyUIBtn;
		tyBtnSendWorkOrderInfo : tyUIBtn;
		tyBtnInsertBrd : tyUIBtn;
		tyBitmapMask : tyUIBitmap;
		tyLyr : tyUILyr;
	END_STRUCT;
END_TYPE

(**)

TYPE
	tyLyrP1023McSetHCommSel : 	STRUCT
		tyBtnSMEMA : tyUIBtn := (bRtLk:=TRUE,bValue:=TRUE);
		tyBtnHermes : tyUIBtn;
		tyLyr : tyUILyr;
	END_STRUCT;
	tyLyrP1023McSetHCommSMEMA : 	STRUCT
		tyDrpDnSMEMAMod : tyUIDrpDn;
		tyBtnGdSig : tyUIBtn;
		tyLyr : tyUILyr := (uiRtStat:=1);
	END_STRUCT;
	tyLyrP1023McSetHCommUSHermes : 	STRUCT
		tyNumSndAliveTm : tyUINum;
		tyNumLaneID : tyUINum;
		tyNumHostPort : tyUINum;
		tyStringHostAddr : tyUIString;
		tyBtnCheckAliveResponse : tyUIBtn;
		tyBtnOverWrite : tyUIBtn;
		tyBtnCmpParam : tyUIBtn;
		tyBtnCmpTypeId : tyUIBtn;
		tyBtnCommand : tyUIBtn;
		tyBtnBoardForecast : tyUIBtn;
		tyBtnQueryBoardInfo : tyUIBtn;
		tyBitmapMask : tyUIBitmap;
		tyLyr : tyUILyr := (uiRtStat:=1);
	END_STRUCT;
	tyLyrP1023McSetHCommDSHermes : 	STRUCT
		tyNumLaneID : tyUINum;
		tyNumSvrPort : tyUINum;
		tyNumSndAliveTm : tyUINum;
		tyBtnCheckAliveResponse : tyUIBtn;
		tyBtnCommand : tyUIBtn;
		tyBtnBoardForecast : tyUIBtn;
		tyBtnSendBoardInfo : tyUIBtn;
		tyBitmapMask : tyUIBitmap;
		tyLyr : tyUILyr := (uiRtStat:=1);
	END_STRUCT;
	tyLyrP1023McSetHCommGen : 	STRUCT
		tyTxtLblUSSel : tyUITxt;
		tyDrpDnUSSel : tyUIDrpDn;
		tyTxtLblDSSel : tyUITxt;
		tyDrpDnDSSel : tyUIDrpDn;
		tyLyr : tyUILyr;
	END_STRUCT;
END_TYPE

(**)

TYPE
	tyLyrP1024McSetAntiGap : 	STRUCT
		tyTxtLftSen : tyUITxt;
		tyTxtRgtSen : tyUITxt;
		tyNumLftSenOff : tyUINum;
		tyNumRgtSenOff : tyUINum;
		tyLyr : tyUILyr;
	END_STRUCT;
END_TYPE

(**)

TYPE
	tyLyrP1026McSetTeach : 	STRUCT
		tyBtnGet : tyUIBtn;
		tyBtnGo : tyUIBtn;
		tyLyr : tyUILyr;
	END_STRUCT;
END_TYPE

(**)

TYPE
	tyLyrP1040ProdSet : 	STRUCT
		tyBtnDelete : tyUIBtn;
		tyBtnSave : tyUIBtn;
		tyNumProdWidth : tyUINum;
		tyNumProdWidth2 : tyUINum;
		tyStringRecipeNm : tyUILString;
		tyStringSearch : tyUILString;
		tyTableRecipe : tyUITable;
		tyDrpDnMcMode : tyUIDrpDn;
		tyDrpDnFlippedBrd : tyUIDrpDn;
		tyTxtDrpDnFlippedBrd : tyUITxt;
		tyTxtMatchCode : tyUITxt;
		tyStringMatchCode : tyUIString;
		tyLyr : tyUILyr;
		tyBtnToXML : tyUIBtn;
		tyBtnFromXML : tyUIBtn;
		tyBtnSort : tyUIBtn;
		tyHotspotShowLRcp : tyUIHotspot;
	END_STRUCT;
END_TYPE

(**)

TYPE
	tyLyrP1050LFSetLdr : 	STRUCT
		tyTable1List : tyUITable1;
		tyBtnEdit : tyUIBtn;
		tyBtnDelete : tyUIBtn;
		tyBtnOnline : tyUIBtn;
		tyBtnOffline : tyUIBtn;
		tyBtnShftUp : tyUIBtn;
		tyBtnShftDwn : tyUIBtn;
		tyNumBeforeOven : tyUINum;
		tyNumBeforeOven2 : tyUINum;
		tyNumAfterOven : tyUINum;
		tyNumAfterOven2 : tyUINum;
		tyLyr : tyUILyr;
	END_STRUCT;
	tyLyrP1050LFSetLdrEdit : 	STRUCT
		tyNumMcNum : tyUINum;
		tyStringIPAddr : tyUIString;
		tyBtnOk : tyUIBtn;
		tyBtnCancel : tyUIBtn;
		tyTxtLblInfoThirdParty : tyUITxt;
		tyLyr : tyUILyr;
	END_STRUCT;
END_TYPE

(**)

TYPE
	tyLyrP1080UsrMgmt : 	STRUCT
		tyBtnEditDetail : tyUIBtn;
		tyBtnEditAccess : tyUIBtn;
		tyBtnNewUsr : tyUIBtn;
		tyBtnDeleteUsr : tyUIBtn;
		tyDrpDnLvl : tyUIDrpDn;
		tyTableList : tyUITable1;
		tyLyr : tyUILyr;
	END_STRUCT;
	tyLyrP1080UsrMgmtAct : 	STRUCT
		tyBtnOk : tyUIBtn;
		tyBtnCancel : tyUIBtn;
		tyStringPw : tyUIString;
		tyStringUsrNm : tyUIString;
		tyDrpDnLvl : tyUIDrpDn;
		tyLyr : tyUILyr;
	END_STRUCT;
END_TYPE

(**)

TYPE
	tyLyrP1081UsrMgmtUsrAccessRgtSel : 	STRUCT
		tyDrpDnLevel : tyUIDrpDn;
		tyLyr : tyUILyr;
	END_STRUCT;
	tyLyrP1081UsrMgmtUsrAccessRgt : 	STRUCT
		tyBtnOps : tyUIBtn;
		tyBtnProdSel : tyUIBtn;
		tyBtnMagSel : tyUIBtn;
		tyBtnMcInfo : tyUIBtn;
		tyBtnAlm : tyUIBtn;
		tyBtnBffrInfo : tyUIBtn;
		tyBtnOvenInfo : tyUIBtn;
		tyBtnMagInfo : tyUIBtn;
		tyBtnLFCtrl : tyUIBtn;
		tyBtnManual : tyUIBtn;
		tyBtnManualFBOnly : tyUIBtn;
		tyBtnSimu : tyUIBtn;
		tyBtnChgParam : tyUIBtn;
		tyBtnLFSet : tyUIBtn;
		tyBtnLang : tyUIBtn;
		tyBtnMcSet : tyUIBtn;
		tyBtnProdSet : tyUIBtn;
		tyBtnMagSet : tyUIBtn;
		tyStringNm : tyUIString;
		tyTxtTitle : tyUITxt;
		tyLyr : tyUILyr;
	END_STRUCT;
END_TYPE

(**)
(*Visu Property*)

TYPE
	tyVisu : 	STRUCT
		uiChgPage : UINT;
		uiCurrPage : UINT;
		uiSSaverTm : UINT;
		uiSSaverRemainTm : UINT;
		usiChgLang : USINT;
		usiCurrLang : USINT;
	END_STRUCT;
	tyKeypad : 	STRUCT
		tyTxtTitle : tyUITxt;
	END_STRUCT;
	tyTxtSnippets : 	STRUCT
		sLibraryNm : STRING[10];
		sUsrMgmtUsrLv1Nm : STRING[80];
		sUsrMgmtUsrLv2Nm : STRING[80];
		sUsrMgmtUsrLv3Nm : STRING[80];
	END_STRUCT;
END_TYPE
```

#### Visu_Layer.var - Change By Project
```iecst
(*2020-10-08*)
(**)
(*Reference Common Layer*)
VAR
	p_tyC0001MotionStd : REFERENCE TO tyLyrC0001MotionStd; (*Motion Standard*)
END_VAR
(**)
VAR
	p_tyC0002FullMask : REFERENCE TO tyLyrC0002FullMask; (*Full Mask*)
END_VAR
(**)
VAR
	p_tyC0003DualMask : REFERENCE TO tyLyrC0003DualMask; (*Dual Mask*)
END_VAR
(**)
VAR
	p_tyC0004Navi : REFERENCE TO tyLyrC0004Navi; (*Navigation*)
END_VAR
(**)
VAR
	p_tyC0005Main : REFERENCE TO tyLyrC0005Main; (*Main*)
END_VAR
(**)
VAR
	p_tyC0006Set : REFERENCE TO tyLyrC0006Set; (*Setting*)
END_VAR
(**)
VAR
	p_tyC0007Notif : REFERENCE TO tyLyrC0007Notif; (*Notification*)
END_VAR
(**)
VAR
	p_tyC0008MsgBox : REFERENCE TO tyLyrC0008MsgBox; (*Message Box*)
END_VAR
(**)
VAR
	p_tyC0009Info : REFERENCE TO tyLyrC0009Info; (*Info*)
END_VAR
(**)
VAR
	p_tyC0010RcyMsg : REFERENCE TO tyLyrC0010RcyMsg; (*Recover Msg*)
END_VAR
(**)
VAR
	p_tyC0011Loading : REFERENCE TO tyLyrC0011Loading; (*Recover Msg*)
END_VAR
(**)
VAR
	p_tyC0012RcpPopUp : REFERENCE TO tyLyrC0012RcpPopUp; (*254 Char Rcp Pop Up Layer*)
END_VAR
(**)
VAR
	p_tyP0000SSaver : REFERENCE TO tyLyrP0000SSaver; (*Screen Saver*)
END_VAR
(*Reference Layer*)
(**)
VAR
	p_tyP0001Startup : REFERENCE TO tyLyrP0001Startup; (*Startup*)
	p_tyP0001Initial : REFERENCE TO tyLyrP0001Initial; (*Startup*)
END_VAR
(**)
VAR
	p_tyP0002Menu : REFERENCE TO tyLyrP0002Menu; (*Menu*)
END_VAR
(**)
VAR
	p_tyP0100Login : REFERENCE TO tyLyrP0100Login; (*Login*)
	p_tyP0100Logout : REFERENCE TO tyLyrP0100Logout; (*Logout*)
END_VAR
(**)
VAR
	p_tyP0200OpsGen : REFERENCE TO tyLyrP0200OpsGen; (*Operation*)
	p_tyP0200OpsUSVSMEMA : REFERENCE TO tyLyrP0200OpsUSVSMEMA; (*Operation*)
	p_tyP0200OpsDSVSMEMA : REFERENCE TO tyLyrP0200OpsDSVSMEMA; (*Operation*)
	p_tyP0200OpsUSVSMEMA1 : REFERENCE TO tyLyrP0200OpsUSVSMEMA1; (*Operation*)
	p_tyP0200OpsDSVSMEMA1 : REFERENCE TO tyLyrP0200OpsDSVSMEMA1; (*Operation*)
	p_tyP0200OpsUSVSMEMA2 : REFERENCE TO tyLyrP0200OpsUSVSMEMA2; (*Operation*)
	p_tyP0200OpsBypsInitConv : REFERENCE TO tyLyrP0200OpsBypsInitConv; (*Operation - Reminder Message*)
END_VAR
(**)
VAR
	p_tyP0201OpsConv : REFERENCE TO tyLyrP0201OpsConv;
	p_tyP0201OpsConvIOMonitor : REFERENCE TO tyLyrP0201OpsConvIOMonitor; (*Operation - IO Monitor*)
	p_tyP0201OpsConvIOMonitorMacSafe : REFERENCE TO tyLyrP0201OpsConvIOMonitorMSafe; (*Operation - IO Monitor*)
	p_tyP0201OpsConvIOMonitorXStd : REFERENCE TO tyLyrP0201OpsConvIOMonitorXStd; (*Operation - IO Monitor*)
	p_tyP0201OpsConvChgParam : REFERENCE TO tyLyrP0201OpsConvChgParam; (*Operation - Change Parameter*)
	p_tyP0201OpsConvBypsInitConv : REFERENCE TO tyLyrP0201OpsConvBypsInitConv; (*Operation - Bypass Init Conv*)
END_VAR
(**)
VAR
	p_tyP0300McInfo : REFERENCE TO tyLyrP0300McInfo; (*Operation*)
END_VAR
(**)
VAR
	p_tyP0400ProdSel : REFERENCE TO tyLyrP0400ProdSel; (*Product Selection*)
	p_tyP0400RcpDet : REFERENCE TO tyLyrP0400RcpDet; (*Product Selection_Recipe Detail*)
END_VAR
(**)
VAR
	p_tyP0600Alm : REFERENCE TO tyLyrP0600Alm; (*Alarm*)
END_VAR
(**)
VAR
	p_tyP0700LFCtrl : REFERENCE TO tyLyrP0700LFCtrl; (*Lead Follow*)
END_VAR
(**)
VAR
	p_tyP0900GenIn : REFERENCE TO tyLyrP0900GenIn; (*General Input*)
END_VAR
(**)
VAR
	p_tyP0910GenOut : REFERENCE TO tyLyrP0910GenOut; (*General Output*)
END_VAR
(**)
VAR
	p_tyP0920MtrNPneuCtrl : REFERENCE TO tyLyrP0920MtrNPneuCtrl; (*Motor And Pneumatic Control*)
END_VAR
(**)
VAR
	p_tyP0921ClampNoRSCom : REFERENCE TO tyLyrP0921ClampNoRSCom; (*Clamp*)
	p_tyP0921ClampNoRSDC : REFERENCE TO tyLyrP0921ClampNoRSDC;
	p_tyP0921ClampNoRSFB : REFERENCE TO tyLyrP0921ClampNoRSFB;
END_VAR
(**)
VAR
	p_tyP0922InletShutterCom : REFERENCE TO tyLyrP0922InletShutterCom; (*Shutter*)
	p_tyP0922InletShutterDC : REFERENCE TO tyLyrP0922InletShutterDC;
	p_tyP0922InletShutterFB : REFERENCE TO tyLyrP0922InletShutterFB;
	p_tyP0922InletShutterDis : REFERENCE TO tyLyrP0922InletShutterDis;
	p_tyP0922OutletShutterCom : REFERENCE TO tyLyrP0922OutletShutterCom;
	p_tyP0922OutletShutterDC : REFERENCE TO tyLyrP0922OutletShutterDC;
	p_tyP0922OutletShutterFB : REFERENCE TO tyLyrP0922OutletShutterFB;
	p_tyP0922OutletShutterDis : REFERENCE TO tyLyrP0922OutletShutterDis;
END_VAR
(**)
VAR
	p_tyP0923StopperCom : REFERENCE TO tyLyrP0923StopperCom; (*Stopper_Comm*)
	p_tyP0923StopperDC : REFERENCE TO tyLyrP0923StopperDC; (*Stopper_DC*)
	p_tyP0923StopperFB : REFERENCE TO tyLyrP0923StopperFB; (*Stopper_FB*)
END_VAR
(**)
VAR
	p_tyP0924Clamp1WithRSCom : REFERENCE TO tyLyrP0924Clamp1WithRSCom; (*Clamp1WithRS&2*)
	p_tyP0924Clamp1WithRSDC : REFERENCE TO tyLyrP0924Clamp1WithRSDC;
	p_tyP0924Clamp1WithRSFB : REFERENCE TO tyLyrP0924Clamp1WithRSFB;
	p_tyP0924Clamp1WithRSDis : REFERENCE TO tyLyrP0924Clamp1WithRSDis;
	p_tyP0924Clamp2WithRSCom : REFERENCE TO tyLyrP0924Clamp2WithRSCom;
	p_tyP0924Clamp2WithRSDC : REFERENCE TO tyLyrP0924Clamp2WithRSDC;
	p_tyP0924Clamp2WithRSFB : REFERENCE TO tyLyrP0924Clamp2WithRSFB;
	p_tyP0924Clamp2WithRSDis : REFERENCE TO tyLyrP0924Clamp2WithRSDis;
	p_tyP0924Clamp3WithRSCom : REFERENCE TO tyLyrP0924Clamp3WithRSCom;
	p_tyP0924Clamp3WithRSDC : REFERENCE TO tyLyrP0924Clamp3WithRSDC;
	p_tyP0924Clamp3WithRSFB : REFERENCE TO tyLyrP0924Clamp3WithRSFB;
	p_tyP0924Clamp3WithRSDis : REFERENCE TO tyLyrP0924Clamp3WithRSDis;
END_VAR
(**)
VAR
	p_tyP0931ConvCom : REFERENCE TO tyLyrP0931ConvCom; (*Conveyor_Com*)
	p_tyP0931ConvDC : REFERENCE TO tyLyrP0931ConvDC; (*Conveyor_DC*)
	p_tyP0931ConvFB : REFERENCE TO tyLyrP0931ConvFB; (*Conveyor_FB*)
END_VAR
(**)
VAR
	p_tyP0931InvCom : REFERENCE TO tyLyrP0931InvCom; (*Invertor_Com*)
	p_tyP0931InvDC : REFERENCE TO tyLyrP0931InvDC; (*Invertor_DC*)
	p_tyP0931InvFB : REFERENCE TO tyLyrP0931InvFB; (*Invertor_FB*)
END_VAR
(**)
VAR
	p_tyP0934AW : REFERENCE TO tyLyrP0934AW; (*Auto Width*)
END_VAR
(**)
VAR
	p_tyP0940CommCtrlUSSMEMA : REFERENCE TO tyLyrP0940CommCtrlUSSMEMA; (*Communication Control_SMEMAUS*)
	p_tyP0940CommCtrlDSSMEMA : REFERENCE TO tyLyrP0940CommCtrlDSSMEMA; (*Communication Control_SMEMADS*)
	p_tyP0940CommCtrlUSSMEMA2 : REFERENCE TO tyLyrP0940CommCtrlUSSMEMA2; (*Communication Control_SMEMAUS*)
END_VAR
(**)
VAR
	p_tyP0950Simu : REFERENCE TO tyLyrP0950Simu; (*Simulation*)
END_VAR
(**)
VAR
	p_tyP1000Lang : REFERENCE TO tyLyrP1000Lang; (*Language And Setup*)
END_VAR
(**)
VAR
	p_tyP1020McSetNavi : REFERENCE TO tyLyrP1020McSetNavi; (*Machine Setting - Navigation*)
END_VAR
(**)
VAR
	p_tyP1021McSetGen : REFERENCE TO tyLyrP1021McSetGen; (*Machine Setting - General*)
	p_tyP1021McSetNetwork : REFERENCE TO tyLyrP1021McSetNetwork;
END_VAR
(**)
VAR
	p_tyP1022McSetVCommSel : REFERENCE TO tyLyrP1022McSetVCommSel; (*Machine Setting - US Commnunication SMEMA*)
	p_tyP1022McSetVCommLF : REFERENCE TO tyLyrP1022McSetVCommLF; (*Machine Setting - US Commnunication SMEMA*)
	p_tyP1022McSetVCommSvy : REFERENCE TO tyLyrP1022McSetVCommSvy;
END_VAR
(**)
VAR
	p_tyP1023McSetHCommUSSel : REFERENCE TO tyLyrP1023McSetHCommSel; (*Machine Setting - Commnunication Selection*)
	p_tyP1023McSetHCommUSSel2 : REFERENCE TO tyLyrP1023McSetHCommSel; (*Machine Setting - Commnunication Selection*)
	p_tyP1023McSetHCommUSSMEMA : REFERENCE TO tyLyrP1023McSetHCommSMEMA; (*Machine Setting - Commnunication SMEMA*)
	p_tyP1023McSetHCommUSSMEMA2 : REFERENCE TO tyLyrP1023McSetHCommSMEMA; (*Machine Setting - Commnunication SMEMA*)
	p_tyP1023McSetHCommUSHermes : REFERENCE TO tyLyrP1023McSetHCommUSHermes; (*Machine Setting - Commnunication Hermes US*)
	p_tyP1023McSetHCommDSSel : REFERENCE TO tyLyrP1023McSetHCommSel; (*Machine Setting - Commnunication Selection*)
	p_tyP1023McSetHCommDSSMEMA : REFERENCE TO tyLyrP1023McSetHCommSMEMA; (*Machine Setting - Commnunication SMEMA*)
	p_tyP1023McSetHCommDSHermes : REFERENCE TO tyLyrP1023McSetHCommDSHermes; (*Machine Setting - Commnunication Hermes DS*)
	p_tyP1023McSetHCommGen : REFERENCE TO tyLyrP1023McSetHCommGen; (*Machine Setting - Commnunication Selection*)
END_VAR
(**)
VAR
	p_tyP1024McSetAntiGap : REFERENCE TO tyLyrP1024McSetAntiGap; (*Machine Setting - Anti Gap Sensor*)
END_VAR
(**)
VAR
	p_tyP1040ProdSet : REFERENCE TO tyLyrP1040ProdSet; (*Product Setting*)
END_VAR
(**)
VAR
	p_tyP1050LFSetLdr : REFERENCE TO tyLyrP1050LFSetLdr; (*Leader Follower Setup*)
	p_tyP1050LFSetLdrEdit : REFERENCE TO tyLyrP1050LFSetLdrEdit; (*Leader Follower Setup - Edit*)
END_VAR
(**)
VAR
	p_tyP1080UsrMgmt : REFERENCE TO tyLyrP1080UsrMgmt; (*User Management*)
	p_tyP1080UsrMgmtAct : REFERENCE TO tyLyrP1080UsrMgmtAct; (*User Management Edit*)
END_VAR
(**)
VAR
	p_tyP1081UsrMgmtUsrAccessRgtSel : REFERENCE TO tyLyrP1081UsrMgmtUsrAccessRgtSel; (*User Management Edit Access*)
	p_tyP1081UsrMgmtUsrAccessRgt : REFERENCE TO tyLyrP1081UsrMgmtUsrAccessRgt; (*User Management Edit Access*)
END_VAR
(**)
(*Reference Visu Property*)
VAR
	p_tyTxtSnippets : REFERENCE TO tyTxtSnippets; (*Text Snippets*)
	p_tyKeypad : REFERENCE TO tyKeypad; (*Keypad*)
	p_tyVisu : REFERENCE TO tyVisu; (*Visualization Properties*)
END_VAR
```

### Startup.typ - Do Not Change!!!
```iecst
(*2019-04-04*)
(**)

TYPE
	eStartupAction :
		(
		StartupActIdle,
		StartupActRun
		);
	eStartupStep :
		(
		StartupStepUsrFolder,
		StartupStepParameter,
		StartupStepGetHWInfo,
		StartupStepLibVer,
		StartupStepRecipe,
		StartupStepUsrMgmt,
		StartupStepBffr,
		StartupStepAlarm,
		StartupStepHermes,
		StartupStepSDOWrite,
		StartupStepSetupUI,
		StartupStepDone
		);
END_TYPE
```

### Startup.var - Change By Project
```iecst
(*2020-09-16*)
(**)
(*Action & State & Status*)
VAR
	p_StartupStat : UDINT;
	p_StartupStatus : UDINT;
	p_StartupStatTxt : UDINT;
END_VAR
(**)
(*Alarm*)
(**)
(*Output*)
VAR
	p_StartupRun : UDINT;
	p_StartupUsrFolderAct : UDINT;
	p_StartupHWInfoAct : UDINT;
	p_StartupLibVerAct : UDINT;
	p_StartupNtParamAct : UDINT;
	p_StartupMcParamAct : UDINT;
	p_StartupProdRcpAct : UDINT;
	p_StartupMpProdRcpAct : UDINT;
	p_StartupUsrMgmtAct : UDINT;
	p_StartupAlarmAct : UDINT;
	p_StartupUIAct : UDINT;
	p_StartupAWAct : UDINT;
	p_StartupHermesAct : UDINT;
	p_StartupRmtHermesAct : UDINT;
	p_StartupUSHermesAct : UDINT;
	p_StartupDSHermesAct : UDINT;
	p_StartupStep : UDINT;
	p_StartupNtSettingsLoadDone : UDINT;
	p_StartupUISettingsLoadDone : UDINT;
	p_StartupStepTxt : UDINT;
	p_StartupGetConfigDone : UDINT;
	p_StartupMismatchSetConfigDone : UDINT;
END_VAR
```

### Program Logical/Startup/Startup (IEC, version 1.00.0) - 1.00.0 - 

#### Init.st - Change By Project
```iecst
(** 2020-09-16 **)
PROGRAM _INIT

	(* Always Change If Project Change *)

	//Pass Address To External Use
	p_StartupStat		:= ADR(eStat);
	p_StartupStatus		:= ADR(eStatus);
	p_StartupStatTxt	:= ADR(sStatTxt);

	//Alarm

	//Output
	p_StartupRun				:= ADR(bRun);
	p_StartupUsrFolderAct		:= ADR(eUsrFolderAct);
	p_StartupHWInfoAct			:= ADR(eHWInfoAct);
	p_StartupLibVerAct			:= ADR(eLibVerAct);
	p_StartupNtParamAct			:= ADR(eNtParamAct);
	p_StartupMcParamAct			:= ADR(eMcParamAct);
	p_StartupProdRcpAct			:= ADR(eProdRcpAct);
	p_StartupMpProdRcpAct		:= ADR(eMpProdRcpAct);
	p_StartupUsrMgmtAct			:= ADR(eUsrMgmtAct);
	p_StartupAlarmAct			:= ADR(eAlarmAct);
	p_StartupUIAct				:= ADR(eUIAct);
	p_StartupAWAct				:= ADR(eAWAct);
	p_StartupHermesAct			:= ADR(eHermesAct);
	p_StartupRmtHermesAct		:= ADR(eRmtHermesAct);
	p_StartupUSHermesAct		:= ADR(eUSHermesAct);
	p_StartupDSHermesAct		:= ADR(eDSHermesAct);
	p_StartupStep				:= ADR(eStartupStep1);
	p_StartupNtSettingsLoadDone	:= ADR(bNtSettingsLoadDone);
	p_StartupUISettingsLoadDone := ADR(bUISettingsLoadDone);
	p_StartupStepTxt			:= ADR(sStepTxt);

	p_StartupGetConfigDone			:= ADR(bGetConfigDone);
	p_StartupMismatchSetConfigDone	:= ADR(bMismatchSetConfigDone);

	(* Always Change If Project Change *)

END_PROGRAM
```

#### Act_InitGlobal.st - Change By Project
```iecst
(** 2020-09-22 **)
ACTION Act_InitGlobal:

	(* Always Change If Project Change *)

	//Pass Data To Link

	//Pass Data To Internal Use
	p_eAct ACCESS p_UIStartupAct;
	p_tyNtParamCurr ACCESS p_NtParamCurr;
	p_tyMcParamCurr ACCESS p_McParamCurr;

	p_bUIMismatchOverWriteConfig ACCESS p_UIMismatchOverWriteConfig;
	p_bUITempAddrFillDone ACCESS p_UITempAddrFillDone;
	p_bUIChgConfigDone ACCESS p_UIIPConfigChgDone;
	p_bUIOverwriteIP ACCESS p_UIOverwriteIP;
	p_bUIOverwriteSubnet ACCESS p_UIOverwriteSubnet;
	p_bUIOverwriteEthMode ACCESS p_UIOverwriteEthMode;

	p_eUsrFolderStat ACCESS p_UsrFolderStat;
	p_eUsrFolderStatus ACCESS p_UsrFolderStatus;

	p_eHWInfoStat ACCESS p_HWInfoStat;
	p_eHWInfoStatus ACCESS p_HWInfoStatus;
	p_sHWInfoIPAddr ACCESS p_HWInfoIPAddr;
	p_sHWInfoSubnetMask ACCESS p_HWInfoSubnetMask;
	p_udiHWInfoEthMode ACCESS p_HWInfoEthMode;

	p_eLibVerStat ACCESS p_LibVerStat;
	p_eLibVerStatus ACCESS p_LibVerStatus;

	p_eNtParamStat ACCESS p_NtParamStat;
	p_eNtParamStatus ACCESS p_NtParamStatus;

	p_eMcParamStat ACCESS p_McParamStat;
	p_eMcParamStatus ACCESS p_McParamStatus;

	p_eProdRcpStat ACCESS p_ProdRcpStat;
	p_eProdRcpStatus ACCESS p_ProdRcpStatus;

	p_eMpProdRcpStat ACCESS p_MpProdRcpStat;
	p_eMpProdRcpStatus ACCESS p_MpProdRcpStatus;

	p_eUsrMgmtStat ACCESS p_UsrMgmtStat;
	p_eUsrMgmtStatus ACCESS p_UsrMgmtStatus;

	p_eAlarmStat ACCESS p_AlarmStat;
	p_eAlarmStatus ACCESS p_AlarmStatus;

	p_eHermesStat ACCESS p_HermesStat;
	p_eHermesStatus ACCESS p_HermesStatus;

	p_eRmtHermesStat ACCESS p_RmtHermesStat;
	p_eRmtHermesStatus ACCESS p_RmtHermesStatus;

	p_eUSHermesStat ACCESS p_USHermesStat;
	p_eUSHermesStatus ACCESS p_USHermesStatus;

	p_eDSHermesStat ACCESS p_DSHermesStat;
	p_eDSHermesStatus ACCESS p_DSHermesStatus;

	p_eAWStat ACCESS p_AWOpenStat;
	p_eAWStatus ACCESS p_AWOpenStatus;

	p_eUIStat ACCESS p_UIStat;
	p_eUIStatus ACCESS p_UIStatus;

	(* Always Change If Project Change *)

END_ACTION
```
